LIN {X 0,Y 470.04,Z 195.084,A -85,B 0,C 180,E1 -7474.395,E2 -7474.395} C_VEL
LIN {X 0,Y 470.295,Z 182.109,A -85,B 0,C 180,E1 -7474.903,E2 -7474.903} C_VEL
LIN {X 0,Y 470.508,Z 169.126,A -85,B 0,C 180,E1 -7475.223,E2 -7475.223} C_VEL
LIN {X 0,Y 471.114,Z 78.667,A -85,B 0,C 180,E1 -7476.612,E2 -7476.612} C_VEL
LIN {X 0,Y 468.567,Z 65.779,A -85,B 0,C 180,E1 -7476.919,E2 -7476.919} C_VEL
LIN {X 0,Y 468.447,Z 59.054,A -85,B 0,C 180,E1 -7478.387,E2 -7478.387} C_VEL
LIN {X 0,Y 467.663,Z 54.233,A -85,B 0,C 180,E1 -7479.515,E2 -7479.515} C_VEL
LIN {X 0,Y 467.656,Z 54.231,A -85,B 0,C 180,E1 -7482.358,E2 -7482.358} C_VEL
LIN {X 0,Y 467.652,Z 54.229,A -85,B 0,C 180,E1 -7485.886,E2 -7485.886} C_VEL
LIN {X 0,Y 467.625,Z 54.231,A -85,B 0,C 180,E1 -7489.308,E2 -7489.308} C_VEL
LIN {X 0,Y 467.536,Z 54.247,A -85,B 0,C 180,E1 -7492.074,E2 -7492.074} C_VEL
LIN {X 0,Y 467.587,Z 54.237,A -85,B 0,C 180,E1 -7494.889,E2 -7494.889} C_VEL
LIN {X 0,Y 467.629,Z 54.234,A -85,B 0,C 180,E1 -7497.769,E2 -7497.769} C_VEL
LIN {X 0,Y 467.57,Z 54.238,A -85,B 0,C 180,E1 -7501.045,E2 -7501.045} C_VEL
LIN {X 0,Y 467.592,Z 54.238,A -85,B 0,C 180,E1 -7504.243,E2 -7504.243} C_VEL
LIN {X 0,Y 467.552,Z 54.242,A -85,B 0,C 180,E1 -7507.187,E2 -7507.187} C_VEL
LIN {X 0,Y 467.58,Z 54.238,A -85,B 0,C 180,E1 -7510.265,E2 -7510.265} C_VEL
LIN {X 0,Y 467.589,Z 54.236,A -85,B 0,C 180,E1 -7512.567,E2 -7512.567} C_VEL
LIN {X 0,Y 467.568,Z 54.241,A -85,B 0,C 180,E1 -7515.053,E2 -7515.053} C_VEL
LIN {X 0,Y 467.592,Z 54.243,A -85,B 0,C 180,E1 -7517.44,E2 -7517.44} C_VEL
LIN {X 0,Y 467.579,Z 54.24,A -85,B 0,C 180,E1 -7520.855,E2 -7520.855} C_VEL
LIN {X 0,Y 467.563,Z 54.239,A -85,B 0,C 180,E1 -7524.261,E2 -7524.261} C_VEL
LIN {X 0,Y 467.586,Z 54.24,A -85,B 0,C 180,E1 -7527.321,E2 -7527.321} C_VEL
LIN {X 0,Y 467.574,Z 54.242,A -85,B 0,C 180,E1 -7530.668,E2 -7530.668} C_VEL
LIN {X 0,Y 467.62,Z 54.235,A -85,B 0,C 180,E1 -7533.2,E2 -7533.2} C_VEL
LIN {X 0,Y 467.596,Z 54.24,A -85,B 0,C 180,E1 -7536.469,E2 -7536.469} C_VEL
LIN {X 0,Y 467.626,Z 54.231,A -85,B 0,C 180,E1 -7539.777,E2 -7539.777} C_VEL
LIN {X 0,Y 467.601,Z 54.242,A -85,B 0,C 180,E1 -7542.507,E2 -7542.507} C_VEL
LIN {X 0,Y 467.611,Z 54.233,A -85,B 0,C 180,E1 -7545.197,E2 -7545.197} C_VEL
LIN {X 0,Y 467.661,Z 54.229,A -85,B 0,C 180,E1 -7547.855,E2 -7547.855} C_VEL
LIN {X 0,Y 467.674,Z 54.225,A -85,B 0,C 180,E1 -7551.357,E2 -7551.357} C_VEL
LIN {X 0,Y 467.742,Z 54.223,A -85,B 0,C 180,E1 -7553.963,E2 -7553.963} C_VEL
LIN {X 0,Y 467.857,Z 54.204,A -85,B 0,C 180,E1 -7557.417,E2 -7557.417} C_VEL
LIN {X 0,Y 467.887,Z 54.205,A -85,B 0,C 180,E1 -7560,E2 -7560} C_VEL
LIN {X 0,Y 467.863,Z 54.202,A -85,B 0,C 180,E1 -7562.583,E2 -7562.583} C_VEL
LIN {X 0,Y 467.72,Z 54.222,A -85,B 0,C 180,E1 -7566.038,E2 -7566.038} C_VEL
LIN {X 0,Y 467.674,Z 54.225,A -85,B 0,C 180,E1 -7568.643,E2 -7568.643} C_VEL
LIN {X 0,Y 467.662,Z 54.227,A -85,B 0,C 180,E1 -7572.145,E2 -7572.145} C_VEL
LIN {X 0,Y 467.644,Z 54.232,A -85,B 0,C 180,E1 -7575.695,E2 -7575.695} C_VEL
LIN {X 0,Y 467.627,Z 54.237,A -85,B 0,C 180,E1 -7579.308,E2 -7579.308} C_VEL
LIN {X 0,Y 467.539,Z 54.242,A -85,B 0,C 180,E1 -7582.074,E2 -7582.074} C_VEL
LIN {X 0,Y 467.589,Z 54.243,A -85,B 0,C 180,E1 -7584.888,E2 -7584.888} C_VEL
LIN {X 0,Y 467.585,Z 54.236,A -85,B 0,C 180,E1 -7587.771,E2 -7587.771} C_VEL
LIN {X 0,Y 467.573,Z 54.242,A -85,B 0,C 180,E1 -7591.045,E2 -7591.045} C_VEL
LIN {X 0,Y 467.581,Z 54.24,A -85,B 0,C 180,E1 -7594.24,E2 -7594.24} C_VEL
LIN {X 0,Y 467.551,Z 54.241,A -85,B 0,C 180,E1 -7597.186,E2 -7597.186} C_VEL
LIN {X 0,Y 467.579,Z 54.243,A -85,B 0,C 180,E1 -7600.265,E2 -7600.265} C_VEL
LIN {X 0,Y 467.59,Z 54.24,A -85,B 0,C 180,E1 -7602.567,E2 -7602.567} C_VEL
LIN {X 0,Y 467.569,Z 54.238,A -85,B 0,C 180,E1 -7605.052,E2 -7605.052} C_VEL
LIN {X 0,Y 467.576,Z 54.239,A -85,B 0,C 180,E1 -7608.597,E2 -7608.597} C_VEL
LIN {X 0,Y 467.565,Z 54.247,A -85,B 0,C 180,E1 -7611.955,E2 -7611.955} C_VEL
LIN {X 0,Y 467.56,Z 54.24,A -85,B 0,C 180,E1 -7615.167,E2 -7615.167} C_VEL
LIN {X 0,Y 467.585,Z 54.238,A -85,B 0,C 180,E1 -7618.26,E2 -7618.26} C_VEL
LIN {X 0,Y 467.579,Z 54.243,A -85,B 0,C 180,E1 -7621.25,E2 -7621.25} C_VEL
LIN {X 0,Y 467.687,Z 54.395,A -85,B 0,C 180,E1 -7623.385,E2 -7623.385} C_VEL
LIN {X 0,Y 469.815,Z 65.941,A -85,B 0,C 180,E1 -7625.425,E2 -7625.425} C_VEL
LIN {X 0,Y 469.107,Z 85.156,A -85,B 0,C 180,E1 -7628.584,E2 -7628.584} C_VEL
LIN {X 0,Y 468.385,Z 105.335,A -85,B 0,C 180,E1 -7631.859,E2 -7631.859} C_VEL
LIN {X 0,Y 468.112,Z 112.972,A -85,B 0,C 180,E1 -7633.09,E2 -7633.09} C_VEL
LIN {X 0,Y 470.906,Z 134.248,A -85,B 0,C 180,E1 -7633.51,E2 -7633.51} C_VEL
LIN {X 0,Y 470.261,Z 221.943,A -85,B 0,C 180,E1 -7634.866,E2 -7634.866} C_VEL
LIN {X 0,Y 469.892,Z 235.212,A -85,B 0,C 180,E1 -7635.242,E2 -7635.242} C_VEL
LIN {X 0,Y 469.459,Z 247.401,A -85,B 0,C 180,E1 -7635.754,E2 -7635.754} C_VEL
LIN {X 0,Y 468.956,Z 259.7,A -85,B 0,C 180,E1 -7636.457,E2 -7636.457} C_VEL
LIN {X 0,Y 468.438,Z 270.965,A -85,B 0,C 180,E1 -7637.293,E2 -7637.293} C_VEL
LIN {X 0,Y 467.941,Z 281.832,A -85,B 0,C 180,E1 -7638.302,E2 -7638.302} C_VEL
LIN {X 0,Y 467.554,Z 291.258,A -85,B 0,C 180,E1 -7639.389,E2 -7639.389} C_VEL
LIN {X 0,Y 467.158,Z 300.369,A -85,B 0,C 180,E1 -7640.693,E2 -7640.693} C_VEL
LIN {X 0,Y 466.938,Z 307.713,A -85,B 0,C 180,E1 -7641.997,E2 -7641.997} C_VEL
LIN {X 0,Y 466.823,Z 312.679,A -85,B 0,C 180,E1 -7643.082,E2 -7643.082} C_VEL
LIN {X 0,Y 466.728,Z 317.498,A -85,B 0,C 180,E1 -7644.383,E2 -7644.383} C_VEL
LIN {X 0,Y 466.659,Z 321.185,A -85,B 0,C 180,E1 -7645.681,E2 -7645.681} C_VEL
LIN {X 0,Y 466.765,Z 323.097,A -85,B 0,C 180,E1 -7646.547,E2 -7646.547} C_VEL
LIN {X 0,Y 466.711,Z 324.536,A -85,B 0,C 180,E1 -7647.411,E2 -7647.411} C_VEL
LIN {X 0,Y 466.699,Z 325.556,A -85,B 0,C 180,E1 -7648.274,E2 -7648.274} C_VEL
LIN {X 0,Y 466.626,Z 326.42,A -85,B 0,C 180,E1 -7650,E2 -7650} C_VEL
LIN {X 0,Y 466.638,Z 326.234,A -85,B 0,C 180,E1 -7650.863,E2 -7650.863} C_VEL
LIN {X 0,Y 466.699,Z 325.64,A -85,B 0,C 180,E1 -7651.726,E2 -7651.726} C_VEL
LIN {X 0,Y 466.747,Z 323.273,A -85,B 0,C 180,E1 -7653.453,E2 -7653.453} C_VEL
LIN {X 0,Y 466.687,Z 320.35,A -85,B 0,C 180,E1 -7654.751,E2 -7654.751} C_VEL
LIN {X 0,Y 466.705,Z 316.398,A -85,B 0,C 180,E1 -7656.051,E2 -7656.051} C_VEL
LIN {X 0,Y 466.853,Z 311.32,A -85,B 0,C 180,E1 -7657.352,E2 -7657.352} C_VEL
LIN {X 0,Y 467.06,Z 304.951,A -85,B 0,C 180,E1 -7658.654,E2 -7658.654} C_VEL
LIN {X 0,Y 467.347,Z 296.995,A -85,B 0,C 180,E1 -7659.959,E2 -7659.959} C_VEL
LIN {X 0,Y 467.829,Z 288.916,A -85,B 0,C 180,E1 -7661.043,E2 -7661.043} C_VEL
LIN {X 0,Y 468.277,Z 279.075,A -85,B 0,C 180,E1 -7662.129,E2 -7662.129} C_VEL
LIN {X 0,Y 468.796,Z 268.113,A -85,B 0,C 180,E1 -7663.106,E2 -7663.106} C_VEL
LIN {X 0,Y 469.397,Z 255.626,A -85,B 0,C 180,E1 -7663.971,E2 -7663.971} C_VEL
LIN {X 0,Y 469.968,Z 243.381,A -85,B 0,C 180,E1 -7664.617,E2 -7664.617} C_VEL
LIN {X 0,Y 470.446,Z 230.499,A -85,B 0,C 180,E1 -7665.1,E2 -7665.1} C_VEL
LIN {X 0,Y 470.769,Z 216.847,A -85,B 0,C 180,E1 -7665.422,E2 -7665.422} C_VEL
LIN {X 0,Y 471.263,Z 132.801,A -85,B 0,C 180,E1 -7666.727,E2 -7666.727} C_VEL
LIN {X 0,Y 468.293,Z 112.618,A -85,B 0,C 180,E1 -7667.179,E2 -7667.179} C_VEL
LIN {X 0,Y 469.033,Z 94.5,A -85,B 0,C 180,E1 -7670.159,E2 -7670.159} C_VEL
LIN {X 0,Y 469.874,Z 75.402,A -85,B 0,C 180,E1 -7673.351,E2 -7673.351} C_VEL
LIN {X 0,Y 470.248,Z 67.22,A -85,B 0,C 180,E1 -7674.738,E2 -7674.738} C_VEL
LIN {X 0,Y 468.091,Z 56.28,A -85,B 0,C 180,E1 -7676.771,E2 -7676.771} C_VEL
LIN {X 0,Y 467.673,Z 54.232,A -85,B 0,C 180,E1 -7677.19,E2 -7677.19} C_VEL
LIN {X 0,Y 467.572,Z 54.239,A -85,B 0,C 180,E1 -7680.734,E2 -7680.734} C_VEL
LIN {X 0,Y 467.572,Z 54.244,A -85,B 0,C 180,E1 -7683.79,E2 -7683.79} C_VEL
LIN {X 0,Y 467.532,Z 54.244,A -85,B 0,C 180,E1 -7686.962,E2 -7686.962} C_VEL
LIN {X 0,Y 467.585,Z 54.237,A -85,B 0,C 180,E1 -7689.955,E2 -7689.955} C_VEL
LIN {X 0,Y 467.589,Z 54.235,A -85,B 0,C 180,E1 -7692.567,E2 -7692.567} C_VEL
LIN {X 0,Y 467.569,Z 54.237,A -85,B 0,C 180,E1 -7695.053,E2 -7695.053} C_VEL
LIN {X 0,Y 467.592,Z 54.238,A -85,B 0,C 180,E1 -7697.44,E2 -7697.44} C_VEL
LIN {X 0,Y 467.563,Z 54.237,A -85,B 0,C 180,E1 -7700.853,E2 -7700.853} C_VEL
LIN {X 0,Y 467.562,Z 54.238,A -85,B 0,C 180,E1 -7704.261,E2 -7704.261} C_VEL
LIN {X 0,Y 467.583,Z 54.243,A -85,B 0,C 180,E1 -7707.321,E2 -7707.321} C_VEL
LIN {X 0,Y 467.574,Z 54.239,A -85,B 0,C 180,E1 -7710.667,E2 -7710.667} C_VEL
LIN {X 0,Y 467.619,Z 54.234,A -85,B 0,C 180,E1 -7713.2,E2 -7713.2} C_VEL
LIN {X 0,Y 467.596,Z 54.239,A -85,B 0,C 180,E1 -7716.468,E2 -7716.468} C_VEL
LIN {X 0,Y 467.626,Z 54.231,A -85,B 0,C 180,E1 -7719.777,E2 -7719.777} C_VEL
LIN {X 0,Y 467.61,Z 54.236,A -85,B 0,C 180,E1 -7722.507,E2 -7722.507} C_VEL
LIN {X 0,Y 467.611,Z 54.234,A -85,B 0,C 180,E1 -7725.196,E2 -7725.196} C_VEL
LIN {X 0,Y 467.661,Z 54.226,A -85,B 0,C 180,E1 -7727.855,E2 -7727.855} C_VEL
LIN {X 0,Y 467.685,Z 54.225,A -85,B 0,C 180,E1 -7731.357,E2 -7731.357} C_VEL
LIN {X 0,Y 467.742,Z 54.218,A -85,B 0,C 180,E1 -7733.962,E2 -7733.962} C_VEL
LIN {X 0,Y 467.856,Z 54.204,A -85,B 0,C 180,E1 -7737.417,E2 -7737.417} C_VEL
LIN {X 0,Y 467.886,Z 54.205,A -85,B 0,C 180,E1 -7740,E2 -7740} C_VEL
LIN {X 0,Y 467.862,Z 54.2,A -85,B 0,C 180,E1 -7742.583,E2 -7742.583} C_VEL
LIN {X 0,Y 467.73,Z 54.221,A -85,B 0,C 180,E1 -7746.037,E2 -7746.037} C_VEL
LIN {X 0,Y 467.673,Z 54.222,A -85,B 0,C 180,E1 -7748.643,E2 -7748.643} C_VEL
LIN {X 0,Y 467.66,Z 54.227,A -85,B 0,C 180,E1 -7752.145,E2 -7752.145} C_VEL
LIN {X 0,Y 467.643,Z 54.232,A -85,B 0,C 180,E1 -7755.695,E2 -7755.695} C_VEL
LIN {X 0,Y 467.625,Z 54.236,A -85,B 0,C 180,E1 -7759.308,E2 -7759.308} C_VEL
LIN {X 0,Y 467.538,Z 54.242,A -85,B 0,C 180,E1 -7762.074,E2 -7762.074} C_VEL
LIN {X 0,Y 467.595,Z 54.243,A -85,B 0,C 180,E1 -7764.888,E2 -7764.888} C_VEL
LIN {X 0,Y 467.583,Z 54.236,A -85,B 0,C 180,E1 -7767.771,E2 -7767.771} C_VEL
LIN {X 0,Y 467.571,Z 54.24,A -85,B 0,C 180,E1 -7771.045,E2 -7771.045} C_VEL
LIN {X 0,Y 467.579,Z 54.241,A -85,B 0,C 180,E1 -7774.24,E2 -7774.24} C_VEL
LIN {X 0,Y 467.545,Z 54.241,A -85,B 0,C 180,E1 -7777.185,E2 -7777.185} C_VEL
LIN {X 0,Y 467.571,Z 54.237,A -85,B 0,C 180,E1 -7780.265,E2 -7780.265} C_VEL
LIN {X 0,Y 467.55,Z 54.247,A -85,B 0,C 180,E1 -7783.745,E2 -7783.745} C_VEL
LIN {X 0,Y 467.549,Z 54.247,A -85,B 0,C 180,E1 -7786.255,E2 -7786.255} C_VEL
LIN {X 0,Y 467.576,Z 54.24,A -85,B 0,C 180,E1 -7788.724,E2 -7788.724} C_VEL
LIN {X 0,Y 467.562,Z 54.246,A -85,B 0,C 180,E1 -7791.955,E2 -7791.955} C_VEL
LIN {X 0,Y 467.558,Z 54.246,A -85,B 0,C 180,E1 -7795.167,E2 -7795.167} C_VEL
LIN {X 0,Y 467.583,Z 54.245,A -85,B 0,C 180,E1 -7798.26,E2 -7798.26} C_VEL
LIN {X 0,Y 467.654,Z 54.399,A -85,B 0,C 180,E1 -7800.207,E2 -7800.207} C_VEL
LIN {X 0,Y 468.798,Z 61.23,A -85,B 0,C 180,E1 -7801.811,E2 -7801.811} C_VEL
LIN {X 0,Y 468.782,Z 66.257,A -85,B 0,C 180,E1 -7802.91,E2 -7802.91} C_VEL
LIN {X 0,Y 471.756,Z 79.365,A -85,B 0,C 180,E1 -7803.245,E2 -7803.245} C_VEL
LIN {X 0,Y 471.132,Z 151.793,A -85,B 0,C 180,E1 -7804.364,E2 -7804.364} C_VEL
LIN {X 0,Y 470.45,Z 157.646,A -85,B 0,C 180,E1 -7804.426,E2 -7804.426} C_VEL
LIN {X 0,Y 464.651,Z 176.593,A -85,B 0,C 180,E1 -7804.553,E2 -7804.553} C_VEL
LIN {X 0,Y 464.096,Z 180.421,A -85,B 0,C 180,E1 -7804.641,E2 -7804.641} C_VEL
LIN {X 0,Y 464.057,Z 182.332,A -85,B 0,C 180,E1 -7804.7,E2 -7804.7} C_VEL
LIN {X 0,Y 463.797,Z 194.305,A -85,B 0,C 180,E1 -7805.165,E2 -7805.165} C_VEL
LIN {X 0,Y 463.318,Z 206.546,A -85,B 0,C 180,E1 -7805.823,E2 -7805.823} C_VEL
LIN {X 0,Y 462.778,Z 217.982,A -85,B 0,C 180,E1 -7806.625,E2 -7806.625} C_VEL
LIN {X 0,Y 462.245,Z 228.376,A -85,B 0,C 180,E1 -7807.542,E2 -7807.542} C_VEL
LIN {X 0,Y 461.773,Z 237.821,A -85,B 0,C 180,E1 -7808.576,E2 -7808.576} C_VEL
LIN {X 0,Y 461.235,Z 246.36,A -85,B 0,C 180,E1 -7809.717,E2 -7809.717} C_VEL
LIN {X 0,Y 460.738,Z 254.387,A -85,B 0,C 180,E1 -7811.038,E2 -7811.038} C_VEL
LIN {X 0,Y 460.447,Z 260.231,A -85,B 0,C 180,E1 -7812.226,E2 -7812.226} C_VEL
LIN {X 0,Y 460.138,Z 265.635,A -85,B 0,C 180,E1 -7813.587,E2 -7813.587} C_VEL
LIN {X 0,Y 459.936,Z 269.802,A -85,B 0,C 180,E1 -7814.944,E2 -7814.944} C_VEL
LIN {X 0,Y 459.797,Z 271.963,A -85,B 0,C 180,E1 -7815.844,E2 -7815.844} C_VEL
LIN {X 0,Y 459.717,Z 273.644,A -85,B 0,C 180,E1 -7816.743,E2 -7816.743} C_VEL
LIN {X 0,Y 459.659,Z 275.394,A -85,B 0,C 180,E1 -7818.107,E2 -7818.107} C_VEL
LIN {X 0,Y 459.611,Z 276.18,A -85,B 0,C 180,E1 -7819.427,E2 -7819.427} C_VEL
LIN {X 0,Y 459.606,Z 275.831,A -85,B 0,C 180,E1 -7821.204,E2 -7821.204} C_VEL
LIN {X 0,Y 459.657,Z 275.064,A -85,B 0,C 180,E1 -7822.091,E2 -7822.091} C_VEL
LIN {X 0,Y 459.784,Z 272.99,A -85,B 0,C 180,E1 -7823.491,E2 -7823.491} C_VEL
LIN {X 0,Y 459.811,Z 270.242,A -85,B 0,C 180,E1 -7824.738,E2 -7824.738} C_VEL
LIN {X 0,Y 460.024,Z 266.325,A -85,B 0,C 180,E1 -7826.058,E2 -7826.058} C_VEL
LIN {X 0,Y 460.127,Z 261.308,A -85,B 0,C 180,E1 -7827.374,E2 -7827.374} C_VEL
LIN {X 0,Y 460.461,Z 254.977,A -85,B 0,C 180,E1 -7828.688,E2 -7828.688} C_VEL
LIN {X 0,Y 460.855,Z 247.091,A -85,B 0,C 180,E1 -7830,E2 -7830} C_VEL
LIN {X 0,Y 461.294,Z 237.315,A -85,B 0,C 180,E1 -7831.31,E2 -7831.31} C_VEL
LIN {X 0,Y 461.816,Z 228.201,A -85,B 0,C 180,E1 -7832.29,E2 -7832.29} C_VEL
LIN {X 0,Y 462.324,Z 218.3,A -85,B 0,C 180,E1 -7833.159,E2 -7833.159} C_VEL
LIN {X 0,Y 462.804,Z 207.555,A -85,B 0,C 180,E1 -7833.918,E2 -7833.918} C_VEL
LIN {X 0,Y 463.122,Z 195.771,A -85,B 0,C 180,E1 -7834.57,E2 -7834.57} C_VEL
LIN {X 0,Y 463.393,Z 182.979,A -85,B 0,C 180,E1 -7835.085,E2 -7835.085} C_VEL
LIN {X 0,Y 463.614,Z 170.316,A -85,B 0,C 180,E1 -7835.409,E2 -7835.409} C_VEL
LIN {X 0,Y 464.301,Z 79.935,A -85,B 0,C 180,E1 -7836.819,E2 -7836.819} C_VEL
LIN {X 0,Y 461.608,Z 66.201,A -85,B 0,C 180,E1 -7837.133,E2 -7837.133} C_VEL
LIN {X 0,Y 461.454,Z 60.029,A -85,B 0,C 180,E1 -7838.496,E2 -7838.496} C_VEL
LIN {X 0,Y 460.612,Z 55.112,A -85,B 0,C 180,E1 -7839.662,E2 -7839.662} C_VEL
LIN {X 0,Y 460.615,Z 55.11,A -85,B 0,C 180,E1 -7842.445,E2 -7842.445} C_VEL
LIN {X 0,Y 460.602,Z 55.108,A -85,B 0,C 180,E1 -7845.998,E2 -7845.998} C_VEL
LIN {X 0,Y 460.573,Z 55.112,A -85,B 0,C 180,E1 -7848.902,E2 -7848.902} C_VEL
LIN {X 0,Y 460.518,Z 55.117,A -85,B 0,C 180,E1 -7851.486,E2 -7851.486} C_VEL
LIN {X 0,Y 460.533,Z 55.121,A -85,B 0,C 180,E1 -7854.333,E2 -7854.333} C_VEL
LIN {X 0,Y 460.591,Z 55.111,A -85,B 0,C 180,E1 -7857.748,E2 -7857.748} C_VEL
LIN {X 0,Y 460.523,Z 55.117,A -85,B 0,C 180,E1 -7861.283,E2 -7861.283} C_VEL
LIN {X 0,Y 460.536,Z 55.115,A -85,B 0,C 180,E1 -7864.506,E2 -7864.506} C_VEL
LIN {X 0,Y 460.53,Z 55.121,A -85,B 0,C 180,E1 -7867.621,E2 -7867.621} C_VEL
LIN {X 0,Y 460.544,Z 55.114,A -85,B 0,C 180,E1 -7870.27,E2 -7870.27} C_VEL
LIN {X 0,Y 460.501,Z 55.124,A -85,B 0,C 180,E1 -7873.376,E2 -7873.376} C_VEL
LIN {X 0,Y 460.501,Z 55.119,A -85,B 0,C 180,E1 -7876.625,E2 -7876.625} C_VEL
LIN {X 0,Y 460.542,Z 55.116,A -85,B 0,C 180,E1 -7879.731,E2 -7879.731} C_VEL
LIN {X 0,Y 460.503,Z 55.119,A -85,B 0,C 180,E1 -7882.524,E2 -7882.524} C_VEL
LIN {X 0,Y 460.55,Z 55.114,A -85,B 0,C 180,E1 -7885.624,E2 -7885.624} C_VEL
LIN {X 0,Y 460.541,Z 55.119,A -85,B 0,C 180,E1 -7888.745,E2 -7888.745} C_VEL
LIN {X 0,Y 460.585,Z 55.109,A -85,B 0,C 180,E1 -7892.254,E2 -7892.254} C_VEL
LIN {X 0,Y 460.562,Z 55.118,A -85,B 0,C 180,E1 -7894.706,E2 -7894.706} C_VEL
LIN {X 0,Y 460.515,Z 55.117,A -85,B 0,C 180,E1 -7897.572,E2 -7897.572} C_VEL
LIN {X 0,Y 460.572,Z 55.115,A -85,B 0,C 180,E1 -7900.385,E2 -7900.385} C_VEL
LIN {X 0,Y 460.609,Z 55.109,A -85,B 0,C 180,E1 -7904.059,E2 -7904.059} C_VEL
LIN {X 0,Y 460.614,Z 55.106,A -85,B 0,C 180,E1 -7907.666,E2 -7907.666} C_VEL
LIN {X 0,Y 460.624,Z 55.103,A -85,B 0,C 180,E1 -7911.224,E2 -7911.224} C_VEL
LIN {X 0,Y 460.707,Z 55.098,A -85,B 0,C 180,E1 -7913.87,E2 -7913.87} C_VEL
LIN {X 0,Y 460.797,Z 55.083,A -85,B 0,C 180,E1 -7917.378,E2 -7917.378} C_VEL
LIN {X 0,Y 460.858,Z 55.08,A -85,B 0,C 180,E1 -7920,E2 -7920} C_VEL
LIN {X 0,Y 460.804,Z 55.081,A -85,B 0,C 180,E1 -7922.623,E2 -7922.623} C_VEL
LIN {X 0,Y 460.685,Z 55.098,A -85,B 0,C 180,E1 -7926.13,E2 -7926.13} C_VEL
LIN {X 0,Y 460.624,Z 55.104,A -85,B 0,C 180,E1 -7928.776,E2 -7928.776} C_VEL
LIN {X 0,Y 460.619,Z 55.104,A -85,B 0,C 180,E1 -7932.445,E2 -7932.445} C_VEL
LIN {X 0,Y 460.606,Z 55.106,A -85,B 0,C 180,E1 -7935.997,E2 -7935.997} C_VEL
LIN {X 0,Y 460.573,Z 55.112,A -85,B 0,C 180,E1 -7939.615,E2 -7939.615} C_VEL
LIN {X 0,Y 460.515,Z 55.118,A -85,B 0,C 180,E1 -7942.429,E2 -7942.429} C_VEL
LIN {X 0,Y 460.553,Z 55.112,A -85,B 0,C 180,E1 -7945.797,E2 -7945.797} C_VEL
LIN {X 0,Y 460.532,Z 55.116,A -85,B 0,C 180,E1 -7948.235,E2 -7948.235} C_VEL
LIN {X 0,Y 460.525,Z 55.117,A -85,B 0,C 180,E1 -7951.283,E2 -7951.283} C_VEL
LIN {X 0,Y 460.527,Z 55.122,A -85,B 0,C 180,E1 -7954.504,E2 -7954.504} C_VEL
LIN {X 0,Y 460.505,Z 55.118,A -85,B 0,C 180,E1 -7957.623,E2 -7957.623} C_VEL
LIN {X 0,Y 460.543,Z 55.12,A -85,B 0,C 180,E1 -7960.269,E2 -7960.269} C_VEL
LIN {X 0,Y 460.5,Z 55.119,A -85,B 0,C 180,E1 -7963.376,E2 -7963.376} C_VEL
LIN {X 0,Y 460.512,Z 55.12,A -85,B 0,C 180,E1 -7966.625,E2 -7966.625} C_VEL
LIN {X 0,Y 460.538,Z 55.118,A -85,B 0,C 180,E1 -7969.732,E2 -7969.732} C_VEL
LIN {X 0,Y 460.5,Z 55.12,A -85,B 0,C 180,E1 -7972.524,E2 -7972.524} C_VEL
LIN {X 0,Y 460.54,Z 55.119,A -85,B 0,C 180,E1 -7975.623,E2 -7975.623} C_VEL
LIN {X 0,Y 460.541,Z 55.114,A -85,B 0,C 180,E1 -7978.744,E2 -7978.744} C_VEL
LIN {X 0,Y 460.585,Z 55.113,A -85,B 0,C 180,E1 -7982.254,E2 -7982.254} C_VEL
LIN {X 0,Y 460.657,Z 55.196,A -85,B 0,C 180,E1 -7983.191,E2 -7983.191} C_VEL
LIN {X 0,Y 462.874,Z 67.26,A -85,B 0,C 180,E1 -7985.356,E2 -7985.356} C_VEL
LIN {X 0,Y 462.084,Z 86.657,A -85,B 0,C 180,E1 -7988.591,E2 -7988.591} C_VEL
LIN {X 0,Y 461.359,Z 106.149,A -85,B 0,C 180,E1 -7991.803,E2 -7991.803} C_VEL
LIN {X 0,Y 461.112,Z 112.556,A -85,B 0,C 180,E1 -7992.852,E2 -7992.852} C_VEL
LIN {X 0,Y 464.049,Z 134.854,A -85,B 0,C 180,E1 -7993.304,E2 -7993.304} C_VEL
LIN {X 0,Y 463.377,Z 221.566,A -85,B 0,C 180,E1 -7994.664,E2 -7994.664} C_VEL
LIN {X 0,Y 462.968,Z 234.835,A -85,B 0,C 180,E1 -7995.045,E2 -7995.045} C_VEL
LIN {X 0,Y 462.499,Z 247.596,A -85,B 0,C 180,E1 -7995.592,E2 -7995.592} C_VEL
LIN {X 0,Y 462.024,Z 258.932,A -85,B 0,C 180,E1 -7996.25,E2 -7996.25} C_VEL
LIN {X 0,Y 461.492,Z 269.96,A -85,B 0,C 180,E1 -7997.072,E2 -7997.072} C_VEL
LIN {X 0,Y 460.934,Z 281.194,A -85,B 0,C 180,E1 -7998.121,E2 -7998.121} C_VEL
LIN {X 0,Y 460.547,Z 290.685,A -85,B 0,C 180,E1 -7999.226,E2 -7999.226} C_VEL
LIN {X 0,Y 460.118,Z 299.831,A -85,B 0,C 180,E1 -8000.549,E2 -8000.549} C_VEL
LIN {X 0,Y 459.884,Z 307.206,A -85,B 0,C 180,E1 -8001.873,E2 -8001.873} C_VEL
LIN {X 0,Y 459.734,Z 312.195,A -85,B 0,C 180,E1 -8002.975,E2 -8002.975} C_VEL
LIN {X 0,Y 459.622,Z 317.037,A -85,B 0,C 180,E1 -8004.296,E2 -8004.296} C_VEL
LIN {X 0,Y 459.574,Z 320.745,A -85,B 0,C 180,E1 -8005.615,E2 -8005.615} C_VEL
LIN {X 0,Y 459.673,Z 322.666,A -85,B 0,C 180,E1 -8006.494,E2 -8006.494} C_VEL
LIN {X 0,Y 459.632,Z 324.124,A -85,B 0,C 180,E1 -8007.371,E2 -8007.371} C_VEL
LIN {X 0,Y 459.635,Z 325.153,A -85,B 0,C 180,E1 -8008.247,E2 -8008.247} C_VEL
LIN {X 0,Y 459.556,Z 326.033,A -85,B 0,C 180,E1 -8010,E2 -8010} C_VEL
LIN {X 0,Y 459.57,Z 325.862,A -85,B 0,C 180,E1 -8010.876,E2 -8010.876} C_VEL
LIN {X 0,Y 459.606,Z 325.275,A -85,B 0,C 180,E1 -8011.752,E2 -8011.752} C_VEL
LIN {X 0,Y 459.631,Z 324.298,A -85,B 0,C 180,E1 -8012.629,E2 -8012.629} C_VEL
LIN {X 0,Y 459.641,Z 322.923,A -85,B 0,C 180,E1 -8013.506,E2 -8013.506} C_VEL
LIN {X 0,Y 459.613,Z 320.02,A -85,B 0,C 180,E1 -8014.824,E2 -8014.824} C_VEL
LIN {X 0,Y 459.635,Z 315.42,A -85,B 0,C 180,E1 -8016.342,E2 -8016.342} C_VEL
LIN {X 0,Y 459.862,Z 309.054,A -85,B 0,C 180,E1 -8017.906,E2 -8017.906} C_VEL
LIN {X 0,Y 460.081,Z 302.225,A -85,B 0,C 180,E1 -8019.23,E2 -8019.23} C_VEL
LIN {X 0,Y 460.47,Z 293.763,A -85,B 0,C 180,E1 -8020.553,E2 -8020.553} C_VEL
LIN {X 0,Y 460.991,Z 285.07,A -85,B 0,C 180,E1 -8021.654,E2 -8021.654} C_VEL
LIN {X 0,Y 461.533,Z 274.017,A -85,B 0,C 180,E1 -8022.791,E2 -8022.791} C_VEL
LIN {X 0,Y 462.12,Z 263.799,A -85,B 0,C 180,E1 -8023.635,E2 -8023.635} C_VEL
LIN {X 0,Y 462.745,Z 252.029,A -85,B 0,C 180,E1 -8024.401,E2 -8024.401} C_VEL
LIN {X 0,Y 463.296,Z 239.822,A -85,B 0,C 180,E1 -8025.001,E2 -8025.001} C_VEL
LIN {X 0,Y 463.755,Z 227.405,A -85,B 0,C 180,E1 -8025.435,E2 -8025.435} C_VEL
LIN {X 0,Y 463.99,Z 214.988,A -85,B 0,C 180,E1 -8025.709,E2 -8025.709} C_VEL
LIN {X 0,Y 464.578,Z 133.953,A -85,B 0,C 180,E1 -8026.981,E2 -8026.981} C_VEL
LIN {X 0,Y 461.333,Z 112.253,A -85,B 0,C 180,E1 -8027.473,E2 -8027.473} C_VEL
LIN {X 0,Y 462.067,Z 95.691,A -85,B 0,C 180,E1 -8030.245,E2 -8030.245} C_VEL
LIN {X 0,Y 462.827,Z 79.337,A -85,B 0,C 180,E1 -8033.018,E2 -8033.018} C_VEL
LIN {X 0,Y 463.369,Z 69.35,A -85,B 0,C 180,E1 -8034.732,E2 -8034.732} C_VEL
LIN {X 0,Y 461.754,Z 60.249,A -85,B 0,C 180,E1 -8036.436,E2 -8036.436} C_VEL
LIN {X 0,Y 460.619,Z 55.111,A -85,B 0,C 180,E1 -8037.448,E2 -8037.448} C_VEL
LIN {X 0,Y 460.513,Z 55.122,A -85,B 0,C 180,E1 -8040.24,E2 -8040.24} C_VEL
LIN {X 0,Y 460.522,Z 55.119,A -85,B 0,C 180,E1 -8043.326,E2 -8043.326} C_VEL
LIN {X 0,Y 460.479,Z 55.125,A -85,B 0,C 180,E1 -8046.529,E2 -8046.529} C_VEL
LIN {X 0,Y 460.535,Z 55.114,A -85,B 0,C 180,E1 -8049.862,E2 -8049.862} C_VEL
LIN {X 0,Y 460.515,Z 55.116,A -85,B 0,C 180,E1 -8052.9,E2 -8052.9} C_VEL
LIN {X 0,Y 460.512,Z 55.121,A -85,B 0,C 180,E1 -8055.831,E2 -8055.831} C_VEL
LIN {X 0,Y 460.534,Z 55.115,A -85,B 0,C 180,E1 -8058.989,E2 -8058.989} C_VEL
LIN {X 0,Y 460.522,Z 55.119,A -85,B 0,C 180,E1 -8061.266,E2 -8061.266} C_VEL
LIN {X 0,Y 460.512,Z 55.117,A -85,B 0,C 180,E1 -8064.554,E2 -8064.554} C_VEL
LIN {X 0,Y 460.533,Z 55.117,A -85,B 0,C 180,E1 -8067.716,E2 -8067.716} C_VEL
LIN {X 0,Y 460.544,Z 55.115,A -85,B 0,C 180,E1 -8070.769,E2 -8070.769} C_VEL
LIN {X 0,Y 460.563,Z 55.109,A -85,B 0,C 180,E1 -8073.735,E2 -8073.735} C_VEL
LIN {X 0,Y 460.549,Z 55.119,A -85,B 0,C 180,E1 -8076.624,E2 -8076.624} C_VEL
LIN {X 0,Y 460.555,Z 55.112,A -85,B 0,C 180,E1 -8079.453,E2 -8079.453} C_VEL
LIN {X 0,Y 460.562,Z 55.115,A -85,B 0,C 180,E1 -8082.23,E2 -8082.23} C_VEL
LIN {X 0,Y 460.57,Z 55.113,A -85,B 0,C 180,E1 -8084.965,E2 -8084.965} C_VEL
LIN {X 0,Y 460.615,Z 55.108,A -85,B 0,C 180,E1 -8088.559,E2 -8088.559} C_VEL
LIN {X 0,Y 460.7,Z 55.097,A -85,B 0,C 180,E1 -8092.108,E2 -8092.108} C_VEL
LIN {X 0,Y 460.699,Z 55.095,A -85,B 0,C 180,E1 -8094.748,E2 -8094.748} C_VEL
LIN {X 0,Y 460.797,Z 55.083,A -85,B 0,C 180,E1 -8097.377,E2 -8097.377} C_VEL
LIN {X 0,Y 460.857,Z 55.081,A -85,B 0,C 180,E1 -8100,E2 -8100} C_VEL
LIN {X 0,Y 460.802,Z 55.079,A -85,B 0,C 180,E1 -8102.622,E2 -8102.622} C_VEL
LIN {X 0,Y 460.696,Z 55.097,A -85,B 0,C 180,E1 -8106.13,E2 -8106.13} C_VEL
LIN {X 0,Y 460.623,Z 55.101,A -85,B 0,C 180,E1 -8108.776,E2 -8108.776} C_VEL
LIN {X 0,Y 460.617,Z 55.105,A -85,B 0,C 180,E1 -8112.445,E2 -8112.445} C_VEL
LIN {X 0,Y 460.604,Z 55.107,A -85,B 0,C 180,E1 -8115.997,E2 -8115.997} C_VEL
LIN {X 0,Y 460.571,Z 55.111,A -85,B 0,C 180,E1 -8119.615,E2 -8119.615} C_VEL
LIN {X 0,Y 460.514,Z 55.119,A -85,B 0,C 180,E1 -8122.428,E2 -8122.428} C_VEL
LIN {X 0,Y 460.552,Z 55.113,A -85,B 0,C 180,E1 -8125.797,E2 -8125.797} C_VEL
LIN {X 0,Y 460.53,Z 55.117,A -85,B 0,C 180,E1 -8128.234,E2 -8128.234} C_VEL
LIN {X 0,Y 460.523,Z 55.117,A -85,B 0,C 180,E1 -8131.283,E2 -8131.283} C_VEL
LIN {X 0,Y 460.524,Z 55.121,A -85,B 0,C 180,E1 -8134.503,E2 -8134.503} C_VEL
LIN {X 0,Y 460.5,Z 55.12,A -85,B 0,C 180,E1 -8137.623,E2 -8137.623} C_VEL
LIN {X 0,Y 460.528,Z 55.11,A -85,B 0,C 180,E1 -8141.012,E2 -8141.012} C_VEL
LIN {X 0,Y 460.514,Z 55.121,A -85,B 0,C 180,E1 -8144.589,E2 -8144.589} C_VEL
LIN {X 0,Y 460.505,Z 55.125,A -85,B 0,C 180,E1 -8147.816,E2 -8147.816} C_VEL
LIN {X 0,Y 460.519,Z 55.122,A -85,B 0,C 180,E1 -8150.136,E2 -8150.136} C_VEL
LIN {X 0,Y 460.473,Z 55.13,A -85,B 0,C 180,E1 -8153.47,E2 -8153.47} C_VEL
LIN {X 0,Y 460.521,Z 55.123,A -85,B 0,C 180,E1 -8156.674,E2 -8156.674} C_VEL
LIN {X 0,Y 460.591,Z 55.305,A -85,B 0,C 180,E1 -8159.983,E2 -8159.983} C_VEL
LIN {X 0,Y 461.913,Z 63.182,A -85,B 0,C 180,E1 -8161.857,E2 -8161.857} C_VEL
LIN {X 0,Y 461.881,Z 66.521,A -85,B 0,C 180,E1 -8162.606,E2 -8162.606} C_VEL
LIN {X 0,Y 465.099,Z 80.549,A -85,B 0,C 180,E1 -8162.979,E2 -8162.979} C_VEL
LIN {X 0,Y 464.19,Z 172.656,A -85,B 0,C 180,E1 -8164.437,E2 -8164.437} C_VEL
LIN {X 0,Y 464.057,Z 182.332,A -85,B 0,C 180,E1 -8164.7,E2 -8164.7} C_VEL
LIN {X 0,Y 463.383,Z 188.041,A -85,B 0,C 180,E1 -8164.872,E2 -8164.872} C_VEL
LIN {X 0,Y 460.395,Z 197.222,A -85,B 0,C 180,E1 -8165.158,E2 -8165.158} C_VEL
LIN {X 0,Y 457.24,Z 206.104,A -85,B 0,C 180,E1 -8165.542,E2 -8165.542} C_VEL
LIN {X 0,Y 456.311,Z 211.34,A -85,B 0,C 180,E1 -8165.863,E2 -8165.863} C_VEL
LIN {X 0,Y 455.712,Z 222.361,A -85,B 0,C 180,E1 -8166.722,E2 -8166.722} C_VEL
LIN {X 0,Y 455.12,Z 233.364,A -85,B 0,C 180,E1 -8167.802,E2 -8167.802} C_VEL
LIN {X 0,Y 454.571,Z 242.586,A -85,B 0,C 180,E1 -8168.933,E2 -8168.933} C_VEL
LIN {X 0,Y 453.992,Z 251.719,A -85,B 0,C 180,E1 -8170.322,E2 -8170.322} C_VEL
LIN {X 0,Y 453.531,Z 259.009,A -85,B 0,C 180,E1 -8171.712,E2 -8171.712} C_VEL
LIN {X 0,Y 453.233,Z 263.882,A -85,B 0,C 180,E1 -8172.865,E2 -8172.865} C_VEL
LIN {X 0,Y 452.994,Z 268.211,A -85,B 0,C 180,E1 -8174.134,E2 -8174.134} C_VEL
LIN {X 0,Y 452.758,Z 272.079,A -85,B 0,C 180,E1 -8175.619,E2 -8175.619} C_VEL
LIN {X 0,Y 452.666,Z 273.822,A -85,B 0,C 180,E1 -8176.533,E2 -8176.533} C_VEL
LIN {X 0,Y 452.573,Z 275.781,A -85,B 0,C 180,E1 -8178.049,E2 -8178.049} C_VEL
LIN {X 0,Y 452.552,Z 276.542,A -85,B 0,C 180,E1 -8179.26,E2 -8179.26} C_VEL
LIN {X 0,Y 452.508,Z 276.286,A -85,B 0,C 180,E1 -8181.065,E2 -8181.065} C_VEL
LIN {X 0,Y 452.554,Z 275.577,A -85,B 0,C 180,E1 -8181.966,E2 -8181.966} C_VEL
LIN {X 0,Y 452.696,Z 273.392,A -85,B 0,C 180,E1 -8183.507,E2 -8183.507} C_VEL
LIN {X 0,Y 452.752,Z 269.774,A -85,B 0,C 180,E1 -8185.102,E2 -8185.102} C_VEL
LIN {X 0,Y 452.999,Z 265.598,A -85,B 0,C 180,E1 -8186.442,E2 -8186.442} C_VEL
LIN {X 0,Y 453.185,Z 259.281,A -85,B 0,C 180,E1 -8188,E2 -8188} C_VEL
LIN {X 0,Y 453.614,Z 252.377,A -85,B 0,C 180,E1 -8189.334,E2 -8189.334} C_VEL
LIN {X 0,Y 454.002,Z 243.76,A -85,B 0,C 180,E1 -8190.665,E2 -8190.665} C_VEL
LIN {X 0,Y 454.448,Z 234.945,A -85,B 0,C 180,E1 -8191.773,E2 -8191.773} C_VEL
LIN {X 0,Y 454.978,Z 225.255,A -85,B 0,C 180,E1 -8192.767,E2 -8192.767} C_VEL
LIN {X 0,Y 455.54,Z 214.598,A -85,B 0,C 180,E1 -8193.649,E2 -8193.649} C_VEL
LIN {X 0,Y 455.996,Z 202.692,A -85,B 0,C 180,E1 -8194.42,E2 -8194.42} C_VEL
LIN {X 0,Y 456.358,Z 190.303,A -85,B 0,C 180,E1 -8195.025,E2 -8195.025} C_VEL
LIN {X 0,Y 456.614,Z 177.301,A -85,B 0,C 180,E1 -8195.465,E2 -8195.465} C_VEL
LIN {X 0,Y 456.805,Z 161.64,A -85,B 0,C 180,E1 -8195.767,E2 -8195.767} C_VEL
LIN {X 0,Y 457.353,Z 80.446,A -85,B 0,C 180,E1 -8197.046,E2 -8197.046} C_VEL
LIN {X 0,Y 454.655,Z 66.487,A -85,B 0,C 180,E1 -8197.383,E2 -8197.383} C_VEL
LIN {X 0,Y 454.51,Z 61.595,A -85,B 0,C 180,E1 -8198.474,E2 -8198.474} C_VEL
LIN {X 0,Y 453.573,Z 55.988,A -85,B 0,C 180,E1 -8199.814,E2 -8199.814} C_VEL
LIN {X 0,Y 453.565,Z 55.989,A -85,B 0,C 180,E1 -8202.529,E2 -8202.529} C_VEL
LIN {X 0,Y 453.546,Z 55.989,A -85,B 0,C 180,E1 -8206.196,E2 -8206.196} C_VEL
LIN {X 0,Y 453.522,Z 55.989,A -85,B 0,C 180,E1 -8209.041,E2 -8209.041} C_VEL
LIN {X 0,Y 453.478,Z 55.996,A -85,B 0,C 180,E1 -8211.836,E2 -8211.836} C_VEL
LIN {X 0,Y 453.503,Z 55.992,A -85,B 0,C 180,E1 -8214.735,E2 -8214.735} C_VEL
LIN {X 0,Y 453.54,Z 55.992,A -85,B 0,C 180,E1 -8217.961,E2 -8217.961} C_VEL
LIN {X 0,Y 453.468,Z 55.997,A -85,B 0,C 180,E1 -8221.525,E2 -8221.525} C_VEL
LIN {X 0,Y 453.491,Z 55.992,A -85,B 0,C 180,E1 -8224.778,E2 -8224.778} C_VEL
LIN {X 0,Y 453.475,Z 55.995,A -85,B 0,C 180,E1 -8228.311,E2 -8228.311} C_VEL
LIN {X 0,Y 453.496,Z 55.991,A -85,B 0,C 180,E1 -8230.609,E2 -8230.609} C_VEL
LIN {X 0,Y 453.457,Z 56,A -85,B 0,C 180,E1 -8233.244,E2 -8233.244} C_VEL
LIN {X 0,Y 453.466,Z 55.999,A -85,B 0,C 180,E1 -8235.779,E2 -8235.779} C_VEL
LIN {X 0,Y 453.482,Z 55.993,A -85,B 0,C 180,E1 -8238.21,E2 -8238.21} C_VEL
LIN {X 0,Y 453.494,Z 55.994,A -85,B 0,C 180,E1 -8240.794,E2 -8240.794} C_VEL
LIN {X 0,Y 453.458,Z 55.997,A -85,B 0,C 180,E1 -8243.918,E2 -8243.918} C_VEL
LIN {X 0,Y 453.486,Z 55.999,A -85,B 0,C 180,E1 -8247.152,E2 -8247.152} C_VEL
LIN {X 0,Y 453.479,Z 55.994,A -85,B 0,C 180,E1 -8250.269,E2 -8250.269} C_VEL
LIN {X 0,Y 453.511,Z 55.992,A -85,B 0,C 180,E1 -8253.294,E2 -8253.294} C_VEL
LIN {X 0,Y 453.506,Z 55.992,A -85,B 0,C 180,E1 -8256.239,E2 -8256.239} C_VEL
LIN {X 0,Y 453.487,Z 55.994,A -85,B 0,C 180,E1 -8259.118,E2 -8259.118} C_VEL
LIN {X 0,Y 453.506,Z 55.992,A -85,B 0,C 180,E1 -8261.944,E2 -8261.944} C_VEL
LIN {X 0,Y 453.545,Z 55.989,A -85,B 0,C 180,E1 -8264.727,E2 -8264.727} C_VEL
LIN {X 0,Y 453.564,Z 55.989,A -85,B 0,C 180,E1 -8268.379,E2 -8268.379} C_VEL
LIN {X 0,Y 453.59,Z 55.98,A -85,B 0,C 180,E1 -8271.087,E2 -8271.087} C_VEL
LIN {X 0,Y 453.674,Z 55.973,A -85,B 0,C 180,E1 -8273.775,E2 -8273.775} C_VEL
LIN {X 0,Y 453.741,Z 55.962,A -85,B 0,C 180,E1 -8277.337,E2 -8277.337} C_VEL
LIN {X 0,Y 453.828,Z 55.956,A -85,B 0,C 180,E1 -8280,E2 -8280} C_VEL
LIN {X 0,Y 453.748,Z 55.96,A -85,B 0,C 180,E1 -8282.663,E2 -8282.663} C_VEL
LIN {X 0,Y 453.651,Z 55.973,A -85,B 0,C 180,E1 -8286.226,E2 -8286.226} C_VEL
LIN {X 0,Y 453.59,Z 55.981,A -85,B 0,C 180,E1 -8288.914,E2 -8288.914} C_VEL
LIN {X 0,Y 453.569,Z 55.982,A -85,B 0,C 180,E1 -8292.529,E2 -8292.529} C_VEL
LIN {X 0,Y 453.549,Z 55.985,A -85,B 0,C 180,E1 -8296.196,E2 -8296.196} C_VEL
LIN {X 0,Y 453.522,Z 55.994,A -85,B 0,C 180,E1 -8299.039,E2 -8299.039} C_VEL
LIN {X 0,Y 453.481,Z 55.994,A -85,B 0,C 180,E1 -8301.836,E2 -8301.836} C_VEL
LIN {X 0,Y 453.505,Z 55.995,A -85,B 0,C 180,E1 -8304.735,E2 -8304.735} C_VEL
LIN {X 0,Y 453.511,Z 55.99,A -85,B 0,C 180,E1 -8307.953,E2 -8307.953} C_VEL
LIN {X 0,Y 453.48,Z 56.001,A -85,B 0,C 180,E1 -8310.759,E2 -8310.759} C_VEL
LIN {X 0,Y 453.472,Z 55.995,A -85,B 0,C 180,E1 -8313.913,E2 -8313.913} C_VEL
LIN {X 0,Y 453.456,Z 55.997,A -85,B 0,C 180,E1 -8317.19,E2 -8317.19} C_VEL
LIN {X 0,Y 453.487,Z 55.992,A -85,B 0,C 180,E1 -8319.45,E2 -8319.45} C_VEL
LIN {X 0,Y 453.48,Z 55.996,A -85,B 0,C 180,E1 -8321.935,E2 -8321.935} C_VEL
LIN {X 0,Y 453.486,Z 55.993,A -85,B 0,C 180,E1 -8325.471,E2 -8325.471} C_VEL
LIN {X 0,Y 453.467,Z 56.002,A -85,B 0,C 180,E1 -8328.207,E2 -8328.207} C_VEL
LIN {X 0,Y 453.453,Z 55.997,A -85,B 0,C 180,E1 -8330.8,E2 -8330.8} C_VEL
LIN {X 0,Y 453.455,Z 56.004,A -85,B 0,C 180,E1 -8333.917,E2 -8333.917} C_VEL
LIN {X 0,Y 453.482,Z 55.994,A -85,B 0,C 180,E1 -8337.151,E2 -8337.151} C_VEL
LIN {X 0,Y 453.478,Z 55.999,A -85,B 0,C 180,E1 -8340.268,E2 -8340.268} C_VEL
LIN {X 0,Y 453.619,Z 56.161,A -85,B 0,C 180,E1 -8343.021,E2 -8343.021} C_VEL
LIN {X 0,Y 455.819,Z 67.843,A -85,B 0,C 180,E1 -8345.156,E2 -8345.156} C_VEL
LIN {X 0,Y 455.512,Z 77.673,A -85,B 0,C 180,E1 -8346.831,E2 -8346.831} C_VEL
LIN {X 0,Y 454.75,Z 95.831,A -85,B 0,C 180,E1 -8349.887,E2 -8349.887} C_VEL
LIN {X 0,Y 454.132,Z 112.19,A -85,B 0,C 180,E1 -8352.616,E2 -8352.616} C_VEL
LIN {X 0,Y 457.167,Z 136.678,A -85,B 0,C 180,E1 -8353.112,E2 -8353.112} C_VEL
LIN {X 0,Y 456.491,Z 221.092,A -85,B 0,C 180,E1 -8354.456,E2 -8354.456} C_VEL
LIN {X 0,Y 456.033,Z 234.389,A -85,B 0,C 180,E1 -8354.84,E2 -8354.84} C_VEL
LIN {X 0,Y 455.579,Z 246.604,A -85,B 0,C 180,E1 -8355.368,E2 -8355.368} C_VEL
LIN {X 0,Y 455.077,Z 258.113,A -85,B 0,C 180,E1 -8356.036,E2 -8356.036} C_VEL
LIN {X 0,Y 454.491,Z 269.875,A -85,B 0,C 180,E1 -8356.925,E2 -8356.925} C_VEL
LIN {X 0,Y 453.937,Z 280.53,A -85,B 0,C 180,E1 -8357.935,E2 -8357.935} C_VEL
LIN {X 0,Y 453.533,Z 290.088,A -85,B 0,C 180,E1 -8359.057,E2 -8359.057} C_VEL
LIN {X 0,Y 453.072,Z 299.276,A -85,B 0,C 180,E1 -8360.401,E2 -8360.401} C_VEL
LIN {X 0,Y 452.814,Z 306.683,A -85,B 0,C 180,E1 -8361.746,E2 -8361.746} C_VEL
LIN {X 0,Y 452.658,Z 311.701,A -85,B 0,C 180,E1 -8362.865,E2 -8362.865} C_VEL
LIN {X 0,Y 452.525,Z 316.947,A -85,B 0,C 180,E1 -8364.324,E2 -8364.324} C_VEL
LIN {X 0,Y 452.495,Z 320.299,A -85,B 0,C 180,E1 -8365.546,E2 -8365.546} C_VEL
LIN {X 0,Y 452.568,Z 322.229,A -85,B 0,C 180,E1 -8366.439,E2 -8366.439} C_VEL
LIN {X 0,Y 452.555,Z 323.708,A -85,B 0,C 180,E1 -8367.33,E2 -8367.33} C_VEL
LIN {X 0,Y 452.544,Z 324.745,A -85,B 0,C 180,E1 -8368.22,E2 -8368.22} C_VEL
LIN {X 0,Y 452.488,Z 325.645,A -85,B 0,C 180,E1 -8370,E2 -8370} C_VEL
LIN {X 0,Y 452.505,Z 325.492,A -85,B 0,C 180,E1 -8370.89,E2 -8370.89} C_VEL
LIN {X 0,Y 452.553,Z 323.945,A -85,B 0,C 180,E1 -8372.67,E2 -8372.67} C_VEL
LIN {X 0,Y 452.536,Z 322.578,A -85,B 0,C 180,E1 -8373.562,E2 -8373.562} C_VEL
LIN {X 0,Y 452.539,Z 319.696,A -85,B 0,C 180,E1 -8374.9,E2 -8374.9} C_VEL
LIN {X 0,Y 452.554,Z 315.493,A -85,B 0,C 180,E1 -8376.331,E2 -8376.331} C_VEL
LIN {X 0,Y 452.72,Z 310.754,A -85,B 0,C 180,E1 -8377.582,E2 -8377.582} C_VEL
LIN {X 0,Y 452.926,Z 304.447,A -85,B 0,C 180,E1 -8378.927,E2 -8378.927} C_VEL
LIN {X 0,Y 453.283,Z 296.578,A -85,B 0,C 180,E1 -8380.271,E2 -8380.271} C_VEL
LIN {X 0,Y 453.916,Z 286.791,A -85,B 0,C 180,E1 -8381.612,E2 -8381.612} C_VEL
LIN {X 0,Y 454.477,Z 276.478,A -85,B 0,C 180,E1 -8382.748,E2 -8382.748} C_VEL
LIN {X 0,Y 455.13,Z 265.223,A -85,B 0,C 180,E1 -8383.734,E2 -8383.734} C_VEL
LIN {X 0,Y 455.733,Z 254.015,A -85,B 0,C 180,E1 -8384.513,E2 -8384.513} C_VEL
LIN {X 0,Y 456.355,Z 242.677,A -85,B 0,C 180,E1 -8385.12,E2 -8385.12} C_VEL
LIN {X 0,Y 456.863,Z 230.762,A -85,B 0,C 180,E1 -8385.588,E2 -8385.588} C_VEL
LIN {X 0,Y 457.215,Z 217.803,A -85,B 0,C 180,E1 -8385.919,E2 -8385.919} C_VEL
LIN {X 0,Y 457.86,Z 134.698,A -85,B 0,C 180,E1 -8387.253,E2 -8387.253} C_VEL
LIN {X 0,Y 454.814,Z 114.421,A -85,B 0,C 180,E1 -8387.72,E2 -8387.72} C_VEL
LIN {X 0,Y 454.384,Z 111.71,A -85,B 0,C 180,E1 -8387.81,E2 -8387.81} C_VEL
LIN {X 0,Y 455.15,Z 95.52,A -85,B 0,C 180,E1 -8390.566,E2 -8390.566} C_VEL
LIN {X 0,Y 456.056,Z 77.834,A -85,B 0,C 180,E1 -8393.62,E2 -8393.62} C_VEL
LIN {X 0,Y 456.393,Z 69.668,A -85,B 0,C 180,E1 -8395.056,E2 -8395.056} C_VEL
LIN {X 0,Y 453.896,Z 57.411,A -85,B 0,C 180,E1 -8397.429,E2 -8397.429} C_VEL
LIN {X 0,Y 453.547,Z 55.992,A -85,B 0,C 180,E1 -8397.744,E2 -8397.744} C_VEL
LIN {X 0,Y 453.479,Z 55.995,A -85,B 0,C 180,E1 -8400.759,E2 -8400.759} C_VEL
LIN {X 0,Y 453.471,Z 56,A -85,B 0,C 180,E1 -8403.913,E2 -8403.913} C_VEL
LIN {X 0,Y 453.455,Z 55.998,A -85,B 0,C 180,E1 -8407.19,E2 -8407.19} C_VEL
LIN {X 0,Y 453.492,Z 55.99,A -85,B 0,C 180,E1 -8409.45,E2 -8409.45} C_VEL
LIN {X 0,Y 453.479,Z 55.997,A -85,B 0,C 180,E1 -8411.935,E2 -8411.935} C_VEL
LIN {X 0,Y 453.487,Z 55.995,A -85,B 0,C 180,E1 -8415.471,E2 -8415.471} C_VEL
LIN {X 0,Y 453.482,Z 55.993,A -85,B 0,C 180,E1 -8418.209,E2 -8418.209} C_VEL
LIN {X 0,Y 453.49,Z 55.99,A -85,B 0,C 180,E1 -8420.794,E2 -8420.794} C_VEL
LIN {X 0,Y 453.457,Z 55.997,A -85,B 0,C 180,E1 -8423.917,E2 -8423.917} C_VEL
LIN {X 0,Y 453.482,Z 55.996,A -85,B 0,C 180,E1 -8427.151,E2 -8427.151} C_VEL
LIN {X 0,Y 453.479,Z 55.991,A -85,B 0,C 180,E1 -8430.268,E2 -8430.268} C_VEL
LIN {X 0,Y 453.508,Z 55.99,A -85,B 0,C 180,E1 -8433.294,E2 -8433.294} C_VEL
LIN {X 0,Y 453.505,Z 55.993,A -85,B 0,C 180,E1 -8436.239,E2 -8436.239} C_VEL
LIN {X 0,Y 453.487,Z 55.995,A -85,B 0,C 180,E1 -8439.118,E2 -8439.118} C_VEL
LIN {X 0,Y 453.514,Z 55.99,A -85,B 0,C 180,E1 -8441.945,E2 -8441.945} C_VEL
LIN {X 0,Y 453.544,Z 55.99,A -85,B 0,C 180,E1 -8444.726,E2 -8444.726} C_VEL
LIN {X 0,Y 453.564,Z 55.985,A -85,B 0,C 180,E1 -8448.379,E2 -8448.379} C_VEL
LIN {X 0,Y 453.656,Z 55.976,A -85,B 0,C 180,E1 -8451.985,E2 -8451.985} C_VEL
LIN {X 0,Y 453.672,Z 55.971,A -85,B 0,C 180,E1 -8454.667,E2 -8454.667} C_VEL
LIN {X 0,Y 453.741,Z 55.962,A -85,B 0,C 180,E1 -8457.337,E2 -8457.337} C_VEL
LIN {X 0,Y 453.827,Z 55.956,A -85,B 0,C 180,E1 -8460,E2 -8460} C_VEL
LIN {X 0,Y 453.747,Z 55.958,A -85,B 0,C 180,E1 -8462.663,E2 -8462.663} C_VEL
LIN {X 0,Y 453.663,Z 55.972,A -85,B 0,C 180,E1 -8466.225,E2 -8466.225} C_VEL
LIN {X 0,Y 453.589,Z 55.978,A -85,B 0,C 180,E1 -8468.913,E2 -8468.913} C_VEL
LIN {X 0,Y 453.567,Z 55.983,A -85,B 0,C 180,E1 -8472.529,E2 -8472.529} C_VEL
LIN {X 0,Y 453.548,Z 55.986,A -85,B 0,C 180,E1 -8476.196,E2 -8476.196} C_VEL
LIN {X 0,Y 453.52,Z 55.991,A -85,B 0,C 180,E1 -8479.039,E2 -8479.039} C_VEL
LIN {X 0,Y 453.48,Z 55.993,A -85,B 0,C 180,E1 -8481.836,E2 -8481.836} C_VEL
LIN {X 0,Y 453.508,Z 55.996,A -85,B 0,C 180,E1 -8484.735,E2 -8484.735} C_VEL
LIN {X 0,Y 453.509,Z 55.989,A -85,B 0,C 180,E1 -8487.953,E2 -8487.953} C_VEL
LIN {X 0,Y 453.478,Z 55.997,A -85,B 0,C 180,E1 -8490.759,E2 -8490.759} C_VEL
LIN {X 0,Y 453.47,Z 55.996,A -85,B 0,C 180,E1 -8493.913,E2 -8493.913} C_VEL
LIN {X 0,Y 453.451,Z 55.997,A -85,B 0,C 180,E1 -8497.19,E2 -8497.19} C_VEL
LIN {X 0,Y 453.495,Z 55.987,A -85,B 0,C 180,E1 -8500.609,E2 -8500.609} C_VEL
LIN {X 0,Y 453.462,Z 56.002,A -85,B 0,C 180,E1 -8504.222,E2 -8504.222} C_VEL
LIN {X 0,Y 453.449,Z 56,A -85,B 0,C 180,E1 -8507.003,E2 -8507.003} C_VEL
LIN {X 0,Y 453.495,Z 55.997,A -85,B 0,C 180,E1 -8509.409,E2 -8509.409} C_VEL
LIN {X 0,Y 453.45,Z 56.001,A -85,B 0,C 180,E1 -8512.81,E2 -8512.81} C_VEL
LIN {X 0,Y 453.469,Z 56.001,A -85,B 0,C 180,E1 -8516.086,E2 -8516.086} C_VEL
LIN {X 0,Y 453.483,Z 56.004,A -85,B 0,C 180,E1 -8519.612,E2 -8519.612} C_VEL
LIN {X 0,Y 453.497,Z 56.16,A -85,B 0,C 180,E1 -8519.736,E2 -8519.736} C_VEL
LIN {X 0,Y 454.956,Z 64.309,A -85,B 0,C 180,E1 -8521.705,E2 -8521.705} C_VEL
LIN {X 0,Y 455.024,Z 67.18,A -85,B 0,C 180,E1 -8522.305,E2 -8522.305} C_VEL
LIN {X 0,Y 458.39,Z 81.483,A -85,B 0,C 180,E1 -8522.696,E2 -8522.696} C_VEL
LIN {X 0,Y 457.431,Z 173.739,A -85,B 0,C 180,E1 -8524.184,E2 -8524.184} C_VEL
LIN {X 0,Y 457.211,Z 187.048,A -85,B 0,C 180,E1 -8524.588,E2 -8524.588} C_VEL
LIN {X 0,Y 456.866,Z 199.253,A -85,B 0,C 180,E1 -8525.133,E2 -8525.133} C_VEL
LIN {X 0,Y 456.311,Z 211.34,A -85,B 0,C 180,E1 -8525.863,E2 -8525.863} C_VEL
LIN {X 0,Y 455.391,Z 216.549,A -85,B 0,C 180,E1 -8526.217,E2 -8526.217} C_VEL
LIN {X 0,Y 452.187,Z 224.756,A -85,B 0,C 180,E1 -8526.797,E2 -8526.797} C_VEL
LIN {X 0,Y 448.987,Z 232.464,A -85,B 0,C 180,E1 -8527.462,E2 -8527.462} C_VEL
LIN {X 0,Y 448.071,Z 236.852,A -85,B 0,C 180,E1 -8527.941,E2 -8527.941} C_VEL
LIN {X 0,Y 447.486,Z 245.388,A -85,B 0,C 180,E1 -8529.065,E2 -8529.065} C_VEL
LIN {X 0,Y 446.993,Z 253.004,A -85,B 0,C 180,E1 -8530.29,E2 -8530.29} C_VEL
LIN {X 0,Y 446.5,Z 259.853,A -85,B 0,C 180,E1 -8531.651,E2 -8531.651} C_VEL
LIN {X 0,Y 446.132,Z 265.487,A -85,B 0,C 180,E1 -8533.056,E2 -8533.056} C_VEL
LIN {X 0,Y 445.858,Z 269.866,A -85,B 0,C 180,E1 -8534.457,E2 -8534.457} C_VEL
LIN {X 0,Y 445.727,Z 272.167,A -85,B 0,C 180,E1 -8535.387,E2 -8535.387} C_VEL
LIN {X 0,Y 445.6,Z 274.004,A -85,B 0,C 180,E1 -8536.315,E2 -8536.315} C_VEL
LIN {X 0,Y 445.495,Z 276.166,A -85,B 0,C 180,E1 -8537.985,E2 -8537.985} C_VEL
LIN {X 0,Y 445.462,Z 276.884,A -85,B 0,C 180,E1 -8539.087,E2 -8539.087} C_VEL
LIN {X 0,Y 445.396,Z 277.018,A -85,B 0,C 180,E1 -8540.004,E2 -8540.004} C_VEL
LIN {X 0,Y 445.47,Z 276.074,A -85,B 0,C 180,E1 -8541.837,E2 -8541.837} C_VEL
LIN {X 0,Y 445.617,Z 273.806,A -85,B 0,C 180,E1 -8543.513,E2 -8543.513} C_VEL
LIN {X 0,Y 445.668,Z 270.502,A -85,B 0,C 180,E1 -8545.024,E2 -8545.024} C_VEL
LIN {X 0,Y 445.911,Z 266.428,A -85,B 0,C 180,E1 -8546.386,E2 -8546.386} C_VEL
LIN {X 0,Y 446.075,Z 261.218,A -85,B 0,C 180,E1 -8547.743,E2 -8547.743} C_VEL
LIN {X 0,Y 446.488,Z 254.668,A -85,B 0,C 180,E1 -8549.098,E2 -8549.098} C_VEL
LIN {X 0,Y 446.91,Z 246.56,A -85,B 0,C 180,E1 -8550.451,E2 -8550.451} C_VEL
LIN {X 0,Y 447.289,Z 238.289,A -85,B 0,C 180,E1 -8551.576,E2 -8551.576} C_VEL
LIN {X 0,Y 447.875,Z 229.221,A -85,B 0,C 180,E1 -8552.586,E2 -8552.586} C_VEL
LIN {X 0,Y 448.428,Z 219.374,A -85,B 0,C 180,E1 -8553.482,E2 -8553.482} C_VEL
LIN {X 0,Y 448.944,Z 208.696,A -85,B 0,C 180,E1 -8554.264,E2 -8554.264} C_VEL
LIN {X 0,Y 449.303,Z 197.006,A -85,B 0,C 180,E1 -8554.935,E2 -8554.935} C_VEL
LIN {X 0,Y 449.582,Z 184.436,A -85,B 0,C 180,E1 -8555.466,E2 -8555.466} C_VEL
LIN {X 0,Y 449.835,Z 172.332,A -85,B 0,C 180,E1 -8555.801,E2 -8555.801} C_VEL
LIN {X 0,Y 450.542,Z 81.543,A -85,B 0,C 180,E1 -8557.264,E2 -8557.264} C_VEL
LIN {X 0,Y 447.678,Z 66.888,A -85,B 0,C 180,E1 -8557.612,E2 -8557.612} C_VEL
LIN {X 0,Y 447.396,Z 61.964,A -85,B 0,C 180,E1 -8558.729,E2 -8558.729} C_VEL
LIN {X 0,Y 446.523,Z 56.867,A -85,B 0,C 180,E1 -8559.97,E2 -8559.97} C_VEL
LIN {X 0,Y 446.523,Z 56.867,A -85,B 0,C 180,E1 -8562.73,E2 -8562.73} C_VEL
LIN {X 0,Y 446.498,Z 56.867,A -85,B 0,C 180,E1 -8566.228,E2 -8566.228} C_VEL
LIN {X 0,Y 446.471,Z 56.867,A -85,B 0,C 180,E1 -8569.303,E2 -8569.303} C_VEL
LIN {X 0,Y 446.42,Z 56.879,A -85,B 0,C 180,E1 -8572.2,E2 -8572.2} C_VEL
LIN {X 0,Y 446.446,Z 56.87,A -85,B 0,C 180,E1 -8575.153,E2 -8575.153} C_VEL
LIN {X 0,Y 446.486,Z 56.871,A -85,B 0,C 180,E1 -8578.179,E2 -8578.179} C_VEL
LIN {X 0,Y 446.421,Z 56.878,A -85,B 0,C 180,E1 -8581.775,E2 -8581.775} C_VEL
LIN {X 0,Y 446.432,Z 56.872,A -85,B 0,C 180,E1 -8584.523,E2 -8584.523} C_VEL
LIN {X 0,Y 446.433,Z 56.874,A -85,B 0,C 180,E1 -8588.082,E2 -8588.082} C_VEL
LIN {X 0,Y 446.429,Z 56.872,A -85,B 0,C 180,E1 -8590.918,E2 -8590.918} C_VEL
LIN {X 0,Y 446.403,Z 56.879,A -85,B 0,C 180,E1 -8593.846,E2 -8593.846} C_VEL
LIN {X 0,Y 446.4,Z 56.875,A -85,B 0,C 180,E1 -8596.404,E2 -8596.404} C_VEL
LIN {X 0,Y 446.429,Z 56.876,A -85,B 0,C 180,E1 -8599.083,E2 -8599.083} C_VEL
LIN {X 0,Y 446.412,Z 56.874,A -85,B 0,C 180,E1 -8602.122,E2 -8602.122} C_VEL
LIN {X 0,Y 446.433,Z 56.874,A -85,B 0,C 180,E1 -8605.477,E2 -8605.477} C_VEL
LIN {X 0,Y 446.42,Z 56.877,A -85,B 0,C 180,E1 -8608.7,E2 -8608.7} C_VEL
LIN {X 0,Y 446.488,Z 56.864,A -85,B 0,C 180,E1 -8611.822,E2 -8611.822} C_VEL
LIN {X 0,Y 446.462,Z 56.874,A -85,B 0,C 180,E1 -8614.848,E2 -8614.848} C_VEL
LIN {X 0,Y 446.453,Z 56.872,A -85,B 0,C 180,E1 -8618.245,E2 -8618.245} C_VEL
LIN {X 0,Y 446.455,Z 56.869,A -85,B 0,C 180,E1 -8621.649,E2 -8621.649} C_VEL
LIN {X 0,Y 446.513,Z 56.868,A -85,B 0,C 180,E1 -8624.48,E2 -8624.48} C_VEL
LIN {X 0,Y 446.522,Z 56.867,A -85,B 0,C 180,E1 -8628.193,E2 -8628.193} C_VEL
LIN {X 0,Y 446.537,Z 56.859,A -85,B 0,C 180,E1 -8630.945,E2 -8630.945} C_VEL
LIN {X 0,Y 446.642,Z 56.848,A -85,B 0,C 180,E1 -8633.676,E2 -8633.676} C_VEL
LIN {X 0,Y 446.688,Z 56.84,A -85,B 0,C 180,E1 -8637.295,E2 -8637.295} C_VEL
LIN {X 0,Y 446.798,Z 56.831,A -85,B 0,C 180,E1 -8640,E2 -8640} C_VEL
LIN {X 0,Y 446.695,Z 56.839,A -85,B 0,C 180,E1 -8642.705,E2 -8642.705} C_VEL
LIN {X 0,Y 446.62,Z 56.849,A -85,B 0,C 180,E1 -8646.324,E2 -8646.324} C_VEL
LIN {X 0,Y 446.537,Z 56.86,A -85,B 0,C 180,E1 -8649.055,E2 -8649.055} C_VEL
LIN {X 0,Y 446.527,Z 56.86,A -85,B 0,C 180,E1 -8652.73,E2 -8652.73} C_VEL
LIN {X 0,Y 446.501,Z 56.863,A -85,B 0,C 180,E1 -8656.227,E2 -8656.227} C_VEL
LIN {X 0,Y 446.473,Z 56.872,A -85,B 0,C 180,E1 -8659.303,E2 -8659.303} C_VEL
LIN {X 0,Y 446.423,Z 56.873,A -85,B 0,C 180,E1 -8662.2,E2 -8662.2} C_VEL
LIN {X 0,Y 446.447,Z 56.874,A -85,B 0,C 180,E1 -8665.153,E2 -8665.153} C_VEL
LIN {X 0,Y 446.454,Z 56.87,A -85,B 0,C 180,E1 -8668.181,E2 -8668.181} C_VEL
LIN {X 0,Y 446.42,Z 56.874,A -85,B 0,C 180,E1 -8671.3,E2 -8671.3} C_VEL
LIN {X 0,Y 446.427,Z 56.879,A -85,B 0,C 180,E1 -8674.523,E2 -8674.523} C_VEL
LIN {X 0,Y 446.417,Z 56.876,A -85,B 0,C 180,E1 -8678.079,E2 -8678.079} C_VEL
LIN {X 0,Y 446.43,Z 56.873,A -85,B 0,C 180,E1 -8680.917,E2 -8680.917} C_VEL
LIN {X 0,Y 446.402,Z 56.878,A -85,B 0,C 180,E1 -8683.846,E2 -8683.846} C_VEL
LIN {X 0,Y 446.401,Z 56.88,A -85,B 0,C 180,E1 -8686.403,E2 -8686.403} C_VEL
LIN {X 0,Y 446.435,Z 56.875,A -85,B 0,C 180,E1 -8689.801,E2 -8689.801} C_VEL
LIN {X 0,Y 446.403,Z 56.876,A -85,B 0,C 180,E1 -8693.254,E2 -8693.254} C_VEL
LIN {X 0,Y 446.451,Z 56.869,A -85,B 0,C 180,E1 -8696.566,E2 -8696.566} C_VEL
LIN {X 0,Y 446.434,Z 56.879,A -85,B 0,C 180,E1 -8699.979,E2 -8699.979} C_VEL
LIN {X 0,Y 446.555,Z 56.937,A -85,B 0,C 180,E1 -8702.812,E2 -8702.812} C_VEL
LIN {X 0,Y 448.942,Z 69.955,A -85,B 0,C 180,E1 -8705.226,E2 -8705.226} C_VEL
LIN {X 0,Y 448.121,Z 88.258,A -85,B 0,C 180,E1 -8708.373,E2 -8708.373} C_VEL
LIN {X 0,Y 447.27,Z 107.744,A -85,B 0,C 180,E1 -8711.683,E2 -8711.683} C_VEL
LIN {X 0,Y 447.104,Z 111.828,A -85,B 0,C 180,E1 -8712.374,E2 -8712.374} C_VEL
LIN {X 0,Y 450.308,Z 137.238,A -85,B 0,C 180,E1 -8712.897,E2 -8712.897} C_VEL
LIN {X 0,Y 449.596,Z 220.524,A -85,B 0,C 180,E1 -8714.24,E2 -8714.24} C_VEL
LIN {X 0,Y 449.124,Z 233.889,A -85,B 0,C 180,E1 -8714.63,E2 -8714.63} C_VEL
LIN {X 0,Y 448.635,Z 246.709,A -85,B 0,C 180,E1 -8715.194,E2 -8715.194} C_VEL
LIN {X 0,Y 448.058,Z 258.885,A -85,B 0,C 180,E1 -8715.929,E2 -8715.929} C_VEL
LIN {X 0,Y 447.425,Z 270.937,A -85,B 0,C 180,E1 -8716.875,E2 -8716.875} C_VEL
LIN {X 0,Y 446.883,Z 280.923,A -85,B 0,C 180,E1 -8717.857,E2 -8717.857} C_VEL
LIN {X 0,Y 446.504,Z 289.465,A -85,B 0,C 180,E1 -8718.883,E2 -8718.883} C_VEL
LIN {X 0,Y 446.001,Z 298.704,A -85,B 0,C 180,E1 -8720.247,E2 -8720.247} C_VEL
LIN {X 0,Y 445.753,Z 306.149,A -85,B 0,C 180,E1 -8721.614,E2 -8721.614} C_VEL
LIN {X 0,Y 445.51,Z 312.974,A -85,B 0,C 180,E1 -8723.205,E2 -8723.205} C_VEL
LIN {X 0,Y 445.466,Z 317.476,A -85,B 0,C 180,E1 -8724.568,E2 -8724.568} C_VEL
LIN {X 0,Y 445.419,Z 319.846,A -85,B 0,C 180,E1 -8725.475,E2 -8725.475} C_VEL
LIN {X 0,Y 445.465,Z 321.786,A -85,B 0,C 180,E1 -8726.382,E2 -8726.382} C_VEL
LIN {X 0,Y 445.48,Z 323.288,A -85,B 0,C 180,E1 -8727.287,E2 -8727.287} C_VEL
LIN {X 0,Y 445.456,Z 324.336,A -85,B 0,C 180,E1 -8728.192,E2 -8728.192} C_VEL
LIN {X 0,Y 445.442,Z 324.991,A -85,B 0,C 180,E1 -8729.096,E2 -8729.096} C_VEL
LIN {X 0,Y 445.422,Z 325.256,A -85,B 0,C 180,E1 -8730,E2 -8730} C_VEL
LIN {X 0,Y 445.441,Z 325.122,A -85,B 0,C 180,E1 -8730.904,E2 -8730.904} C_VEL
LIN {X 0,Y 445.476,Z 323.596,A -85,B 0,C 180,E1 -8732.713,E2 -8732.713} C_VEL
LIN {X 0,Y 445.433,Z 322.238,A -85,B 0,C 180,E1 -8733.618,E2 -8733.618} C_VEL
LIN {X 0,Y 445.465,Z 319.378,A -85,B 0,C 180,E1 -8734.978,E2 -8734.978} C_VEL
LIN {X 0,Y 445.455,Z 315.49,A -85,B 0,C 180,E1 -8736.341,E2 -8736.341} C_VEL
LIN {X 0,Y 445.67,Z 310.487,A -85,B 0,C 180,E1 -8737.703,E2 -8737.703} C_VEL
LIN {X 0,Y 445.892,Z 304.211,A -85,B 0,C 180,E1 -8739.069,E2 -8739.069} C_VEL
LIN {X 0,Y 446.27,Z 296.395,A -85,B 0,C 180,E1 -8740.434,E2 -8740.434} C_VEL
LIN {X 0,Y 446.939,Z 286.652,A -85,B 0,C 180,E1 -8741.796,E2 -8741.796} C_VEL
LIN {X 0,Y 447.496,Z 277.187,A -85,B 0,C 180,E1 -8742.871,E2 -8742.871} C_VEL
LIN {X 0,Y 448.126,Z 266.674,A -85,B 0,C 180,E1 -8743.837,E2 -8743.837} C_VEL
LIN {X 0,Y 448.876,Z 254.147,A -85,B 0,C 180,E1 -8744.74,E2 -8744.74} C_VEL
LIN {X 0,Y 449.542,Z 241.819,A -85,B 0,C 180,E1 -8745.413,E2 -8745.413} C_VEL
LIN {X 0,Y 450.13,Z 229.648,A -85,B 0,C 180,E1 -8745.886,E2 -8745.886} C_VEL
LIN {X 0,Y 450.474,Z 216.232,A -85,B 0,C 180,E1 -8746.222,E2 -8746.222} C_VEL
LIN {X 0,Y 451.124,Z 135.289,A -85,B 0,C 180,E1 -8747.539,E2 -8747.539} C_VEL
LIN {X 0,Y 447.89,Z 114.019,A -85,B 0,C 180,E1 -8748.042,E2 -8748.042} C_VEL
LIN {X 0,Y 447.465,Z 111.469,A -85,B 0,C 180,E1 -8748.106,E2 -8748.106} C_VEL
LIN {X 0,Y 448.23,Z 95.36,A -85,B 0,C 180,E1 -8750.898,E2 -8750.898} C_VEL
LIN {X 0,Y 449.063,Z 80.424,A -85,B 0,C 180,E1 -8753.521,E2 -8753.521} C_VEL
LIN {X 0,Y 449.553,Z 72.276,A -85,B 0,C 180,E1 -8754.967,E2 -8754.967} C_VEL
LIN {X 0,Y 448.062,Z 63.797,A -85,B 0,C 180,E1 -8756.611,E2 -8756.611} C_VEL
LIN {X 0,Y 446.49,Z 56.871,A -85,B 0,C 180,E1 -8758.006,E2 -8758.006} C_VEL
LIN {X 0,Y 446.418,Z 56.874,A -85,B 0,C 180,E1 -8761.3,E2 -8761.3} C_VEL
LIN {X 0,Y 446.426,Z 56.877,A -85,B 0,C 180,E1 -8764.524,E2 -8764.524} C_VEL
LIN {X 0,Y 446.419,Z 56.877,A -85,B 0,C 180,E1 -8768.079,E2 -8768.079} C_VEL
LIN {X 0,Y 446.43,Z 56.872,A -85,B 0,C 180,E1 -8770.918,E2 -8770.918} C_VEL
LIN {X 0,Y 446.403,Z 56.878,A -85,B 0,C 180,E1 -8773.846,E2 -8773.846} C_VEL
LIN {X 0,Y 446.401,Z 56.874,A -85,B 0,C 180,E1 -8776.404,E2 -8776.404} C_VEL
LIN {X 0,Y 446.43,Z 56.873,A -85,B 0,C 180,E1 -8779.082,E2 -8779.082} C_VEL
LIN {X 0,Y 446.411,Z 56.873,A -85,B 0,C 180,E1 -8782.121,E2 -8782.121} C_VEL
LIN {X 0,Y 446.426,Z 56.874,A -85,B 0,C 180,E1 -8785.477,E2 -8785.477} C_VEL
LIN {X 0,Y 446.419,Z 56.877,A -85,B 0,C 180,E1 -8788.7,E2 -8788.7} C_VEL
LIN {X 0,Y 446.488,Z 56.866,A -85,B 0,C 180,E1 -8791.821,E2 -8791.821} C_VEL
LIN {X 0,Y 446.453,Z 56.872,A -85,B 0,C 180,E1 -8794.847,E2 -8794.847} C_VEL
LIN {X 0,Y 446.452,Z 56.869,A -85,B 0,C 180,E1 -8798.245,E2 -8798.245} C_VEL
LIN {X 0,Y 446.46,Z 56.868,A -85,B 0,C 180,E1 -8801.649,E2 -8801.649} C_VEL
LIN {X 0,Y 446.512,Z 56.866,A -85,B 0,C 180,E1 -8804.48,E2 -8804.48} C_VEL
LIN {X 0,Y 446.522,Z 56.86,A -85,B 0,C 180,E1 -8808.193,E2 -8808.193} C_VEL
LIN {X 0,Y 446.604,Z 56.854,A -85,B 0,C 180,E1 -8811.858,E2 -8811.858} C_VEL
LIN {X 0,Y 446.647,Z 56.847,A -85,B 0,C 180,E1 -8814.583,E2 -8814.583} C_VEL
LIN {X 0,Y 446.667,Z 56.841,A -85,B 0,C 180,E1 -8818.197,E2 -8818.197} C_VEL
LIN {X 0,Y 446.797,Z 56.832,A -85,B 0,C 180,E1 -8820,E2 -8820} C_VEL
LIN {X 0,Y 446.693,Z 56.837,A -85,B 0,C 180,E1 -8822.705,E2 -8822.705} C_VEL
LIN {X 0,Y 446.633,Z 56.848,A -85,B 0,C 180,E1 -8826.324,E2 -8826.324} C_VEL
LIN {X 0,Y 446.536,Z 56.857,A -85,B 0,C 180,E1 -8829.055,E2 -8829.055} C_VEL
LIN {X 0,Y 446.525,Z 56.861,A -85,B 0,C 180,E1 -8832.73,E2 -8832.73} C_VEL
LIN {X 0,Y 446.499,Z 56.864,A -85,B 0,C 180,E1 -8836.227,E2 -8836.227} C_VEL
LIN {X 0,Y 446.471,Z 56.87,A -85,B 0,C 180,E1 -8839.303,E2 -8839.303} C_VEL
LIN {X 0,Y 446.421,Z 56.873,A -85,B 0,C 180,E1 -8842.199,E2 -8842.199} C_VEL
LIN {X 0,Y 446.448,Z 56.873,A -85,B 0,C 180,E1 -8845.153,E2 -8845.153} C_VEL
LIN {X 0,Y 446.452,Z 56.87,A -85,B 0,C 180,E1 -8848.181,E2 -8848.181} C_VEL
LIN {X 0,Y 446.418,Z 56.874,A -85,B 0,C 180,E1 -8851.3,E2 -8851.3} C_VEL
LIN {X 0,Y 446.425,Z 56.877,A -85,B 0,C 180,E1 -8854.523,E2 -8854.523} C_VEL
LIN {X 0,Y 446.413,Z 56.879,A -85,B 0,C 180,E1 -8858.078,E2 -8858.078} C_VEL
LIN {X 0,Y 446.42,Z 56.867,A -85,B 0,C 180,E1 -8861.392,E2 -8861.392} C_VEL
LIN {X 0,Y 446.451,Z 56.872,A -85,B 0,C 180,E1 -8865.104,E2 -8865.104} C_VEL
LIN {X 0,Y 446.42,Z 56.876,A -85,B 0,C 180,E1 -8868.608,E2 -8868.608} C_VEL
LIN {X 0,Y 446.411,Z 56.88,A -85,B 0,C 180,E1 -8871.921,E2 -8871.921} C_VEL
LIN {X 0,Y 446.424,Z 56.88,A -85,B 0,C 180,E1 -8875.476,E2 -8875.476} C_VEL
LIN {X 0,Y 446.418,Z 56.883,A -85,B 0,C 180,E1 -8878.7,E2 -8878.7} C_VEL
LIN {X 0,Y 446.46,Z 57.061,A -85,B 0,C 180,E1 -8879.491,E2 -8879.491} C_VEL
LIN {X 0,Y 448.006,Z 65.082,A -85,B 0,C 180,E1 -8881.46,E2 -8881.46} C_VEL
LIN {X 0,Y 448.098,Z 67.354,A -85,B 0,C 180,E1 -8881.977,E2 -8881.977} C_VEL
LIN {X 0,Y 451.786,Z 82.761,A -85,B 0,C 180,E1 -8882.412,E2 -8882.412} C_VEL
LIN {X 0,Y 450.71,Z 173.707,A -85,B 0,C 180,E1 -8883.895,E2 -8883.895} C_VEL
LIN {X 0,Y 450.461,Z 187.425,A -85,B 0,C 180,E1 -8884.314,E2 -8884.314} C_VEL
LIN {X 0,Y 450.071,Z 200.555,A -85,B 0,C 180,E1 -8884.916,E2 -8884.916} C_VEL
LIN {X 0,Y 449.486,Z 212.233,A -85,B 0,C 180,E1 -8885.645,E2 -8885.645} C_VEL
LIN {X 0,Y 448.813,Z 223.948,A -85,B 0,C 180,E1 -8886.587,E2 -8886.587} C_VEL
LIN {X 0,Y 448.256,Z 233.476,A -85,B 0,C 180,E1 -8887.546,E2 -8887.546} C_VEL
LIN {X 0,Y 448.071,Z 236.852,A -85,B 0,C 180,E1 -8887.941,E2 -8887.941} C_VEL
LIN {X 0,Y 447.147,Z 241.13,A -85,B 0,C 180,E1 -8888.451,E2 -8888.451} C_VEL
LIN {X 0,Y 443.89,Z 247.819,A -85,B 0,C 180,E1 -8889.296,E2 -8889.296} C_VEL
LIN {X 0,Y 440.623,Z 253.911,A -85,B 0,C 180,E1 -8890.217,E2 -8890.217} C_VEL
LIN {X 0,Y 439.697,Z 257.246,A -85,B 0,C 180,E1 -8890.84,E2 -8890.84} C_VEL
LIN {X 0,Y 439.28,Z 263.64,A -85,B 0,C 180,E1 -8892.303,E2 -8892.303} C_VEL
LIN {X 0,Y 438.921,Z 269.021,A -85,B 0,C 180,E1 -8893.888,E2 -8893.888} C_VEL
LIN {X 0,Y 438.703,Z 272.258,A -85,B 0,C 180,E1 -8895.148,E2 -8895.148} C_VEL
LIN {X 0,Y 438.554,Z 274.165,A -85,B 0,C 180,E1 -8896.091,E2 -8896.091} C_VEL
LIN {X 0,Y 438.473,Z 275.596,A -85,B 0,C 180,E1 -8897.033,E2 -8897.033} C_VEL
LIN {X 0,Y 438.422,Z 276.597,A -85,B 0,C 180,E1 -8897.972,E2 -8897.972} C_VEL
LIN {X 0,Y 438.375,Z 277.204,A -85,B 0,C 180,E1 -8898.908,E2 -8898.908} C_VEL
LIN {X 0,Y 438.325,Z 277.418,A -85,B 0,C 180,E1 -8899.842,E2 -8899.842} C_VEL
LIN {X 0,Y 438.331,Z 277.191,A -85,B 0,C 180,E1 -8900.774,E2 -8900.774} C_VEL
LIN {X 0,Y 438.457,Z 275.561,A -85,B 0,C 180,E1 -8902.633,E2 -8902.633} C_VEL
LIN {X 0,Y 438.544,Z 274.147,A -85,B 0,C 180,E1 -8903.559,E2 -8903.559} C_VEL
LIN {X 0,Y 438.589,Z 271.216,A -85,B 0,C 180,E1 -8904.944,E2 -8904.944} C_VEL
LIN {X 0,Y 438.828,Z 267.241,A -85,B 0,C 180,E1 -8906.327,E2 -8906.327} C_VEL
LIN {X 0,Y 439.009,Z 262.145,A -85,B 0,C 180,E1 -8907.706,E2 -8907.706} C_VEL
LIN {X 0,Y 439.391,Z 255.721,A -85,B 0,C 180,E1 -8909.084,E2 -8909.084} C_VEL
LIN {X 0,Y 439.841,Z 247.748,A -85,B 0,C 180,E1 -8910.458,E2 -8910.458} C_VEL
LIN {X 0,Y 440.238,Z 239.633,A -85,B 0,C 180,E1 -8911.601,E2 -8911.601} C_VEL
LIN {X 0,Y 440.852,Z 230.767,A -85,B 0,C 180,E1 -8912.627,E2 -8912.627} C_VEL
LIN {X 0,Y 441.383,Z 221.22,A -85,B 0,C 180,E1 -8913.538,E2 -8913.538} C_VEL
LIN {X 0,Y 441.934,Z 210.942,A -85,B 0,C 180,E1 -8914.332,E2 -8914.332} C_VEL
LIN {X 0,Y 442.366,Z 198.68,A -85,B 0,C 180,E1 -8915.07,E2 -8915.07} C_VEL
LIN {X 0,Y 442.664,Z 185.814,A -85,B 0,C 180,E1 -8915.638,E2 -8915.638} C_VEL
LIN {X 0,Y 442.943,Z 173.172,A -85,B 0,C 180,E1 -8916.005,E2 -8916.005} C_VEL
LIN {X 0,Y 443.783,Z 83.037,A -85,B 0,C 180,E1 -8917.479,E2 -8917.479} C_VEL
LIN {X 0,Y 440.716,Z 67.161,A -85,B 0,C 180,E1 -8917.877,E2 -8917.877} C_VEL
LIN {X 0,Y 440.153,Z 61.503,A -85,B 0,C 180,E1 -8919.188,E2 -8919.188} C_VEL
LIN {X 0,Y 439.463,Z 57.747,A -85,B 0,C 180,E1 -8920.132,E2 -8920.132} C_VEL
LIN {X 0,Y 439.467,Z 57.745,A -85,B 0,C 180,E1 -8922.938,E2 -8922.938} C_VEL
LIN {X 0,Y 439.449,Z 57.747,A -85,B 0,C 180,E1 -8926.349,E2 -8926.349} C_VEL
LIN {X 0,Y 439.404,Z 57.747,A -85,B 0,C 180,E1 -8929.626,E2 -8929.626} C_VEL
LIN {X 0,Y 439.366,Z 57.755,A -85,B 0,C 180,E1 -8932.576,E2 -8932.576} C_VEL
LIN {X 0,Y 439.399,Z 57.749,A -85,B 0,C 180,E1 -8935.586,E2 -8935.586} C_VEL
LIN {X 0,Y 439.419,Z 57.746,A -85,B 0,C 180,E1 -8938.674,E2 -8938.674} C_VEL
LIN {X 0,Y 439.372,Z 57.757,A -85,B 0,C 180,E1 -8942.031,E2 -8942.031} C_VEL
LIN {X 0,Y 439.398,Z 57.75,A -85,B 0,C 180,E1 -8945.341,E2 -8945.341} C_VEL
LIN {X 0,Y 439.393,Z 57.748,A -85,B 0,C 180,E1 -8948.594,E2 -8948.594} C_VEL
LIN {X 0,Y 439.391,Z 57.752,A -85,B 0,C 180,E1 -8951.257,E2 -8951.257} C_VEL
LIN {X 0,Y 439.402,Z 57.748,A -85,B 0,C 180,E1 -8954.73,E2 -8954.73} C_VEL
LIN {X 0,Y 439.398,Z 57.75,A -85,B 0,C 180,E1 -8957.796,E2 -8957.796} C_VEL
LIN {X 0,Y 439.413,Z 57.746,A -85,B 0,C 180,E1 -8960.226,E2 -8960.226} C_VEL
LIN {X 0,Y 439.377,Z 57.752,A -85,B 0,C 180,E1 -8963.713,E2 -8963.713} C_VEL
LIN {X 0,Y 439.377,Z 57.758,A -85,B 0,C 180,E1 -8967.054,E2 -8967.054} C_VEL
LIN {X 0,Y 439.386,Z 57.75,A -85,B 0,C 180,E1 -8970.274,E2 -8970.274} C_VEL
LIN {X 0,Y 439.432,Z 57.745,A -85,B 0,C 180,E1 -8973.397,E2 -8973.397} C_VEL
LIN {X 0,Y 439.391,Z 57.753,A -85,B 0,C 180,E1 -8976.43,E2 -8976.43} C_VEL
LIN {X 0,Y 439.392,Z 57.749,A -85,B 0,C 180,E1 -8979.397,E2 -8979.397} C_VEL
LIN {X 0,Y 439.429,Z 57.749,A -85,B 0,C 180,E1 -8982.31,E2 -8982.31} C_VEL
LIN {X 0,Y 439.452,Z 57.741,A -85,B 0,C 180,E1 -8985.174,E2 -8985.174} C_VEL
LIN {X 0,Y 439.488,Z 57.74,A -85,B 0,C 180,E1 -8988.002,E2 -8988.002} C_VEL
LIN {X 0,Y 439.536,Z 57.733,A -85,B 0,C 180,E1 -8991.726,E2 -8991.726} C_VEL
LIN {X 0,Y 439.622,Z 57.722,A -85,B 0,C 180,E1 -8994.496,E2 -8994.496} C_VEL
LIN {X 0,Y 439.638,Z 57.722,A -85,B 0,C 180,E1 -8998.168,E2 -8998.168} C_VEL
LIN {X 0,Y 439.768,Z 57.707,A -85,B 0,C 180,E1 -9000,E2 -9000} C_VEL
LIN {X 0,Y 439.644,Z 57.717,A -85,B 0,C 180,E1 -9002.749,E2 -9002.749} C_VEL
LIN {X 0,Y 439.571,Z 57.726,A -85,B 0,C 180,E1 -9006.426,E2 -9006.426} C_VEL
LIN {X 0,Y 439.5,Z 57.738,A -85,B 0,C 180,E1 -9009.202,E2 -9009.202} C_VEL
LIN {X 0,Y 439.471,Z 57.741,A -85,B 0,C 180,E1 -9012.938,E2 -9012.938} C_VEL
LIN {X 0,Y 439.451,Z 57.741,A -85,B 0,C 180,E1 -9016.348,E2 -9016.348} C_VEL
LIN {X 0,Y 439.407,Z 57.749,A -85,B 0,C 180,E1 -9019.626,E2 -9019.626} C_VEL
LIN {X 0,Y 439.369,Z 57.753,A -85,B 0,C 180,E1 -9022.575,E2 -9022.575} C_VEL
LIN {X 0,Y 439.385,Z 57.75,A -85,B 0,C 180,E1 -9025.586,E2 -9025.586} C_VEL
LIN {X 0,Y 439.405,Z 57.752,A -85,B 0,C 180,E1 -9028.675,E2 -9028.675} C_VEL
LIN {X 0,Y 439.373,Z 57.752,A -85,B 0,C 180,E1 -9032.03,E2 -9032.03} C_VEL
LIN {X 0,Y 439.396,Z 57.748,A -85,B 0,C 180,E1 -9035.34,E2 -9035.34} C_VEL
LIN {X 0,Y 439.379,Z 57.756,A -85,B 0,C 180,E1 -9038.596,E2 -9038.596} C_VEL
LIN {X 0,Y 439.392,Z 57.748,A -85,B 0,C 180,E1 -9041.257,E2 -9041.257} C_VEL
LIN {X 0,Y 439.402,Z 57.749,A -85,B 0,C 180,E1 -9044.729,E2 -9044.729} C_VEL
LIN {X 0,Y 439.388,Z 57.752,A -85,B 0,C 180,E1 -9047.794,E2 -9047.794} C_VEL
LIN {X 0,Y 439.392,Z 57.754,A -85,B 0,C 180,E1 -9050.223,E2 -9050.223} C_VEL
LIN {X 0,Y 439.375,Z 57.755,A -85,B 0,C 180,E1 -9053.712,E2 -9053.712} C_VEL
LIN {X 0,Y 439.374,Z 57.751,A -85,B 0,C 180,E1 -9057.054,E2 -9057.054} C_VEL
LIN {X 0,Y 439.385,Z 57.755,A -85,B 0,C 180,E1 -9060.274,E2 -9060.274} C_VEL
LIN {X 0,Y 439.517,Z 57.883,A -85,B 0,C 180,E1 -9062.631,E2 -9062.631} C_VEL
LIN {X 0,Y 441.915,Z 70.563,A -85,B 0,C 180,E1 -9065.027,E2 -9065.027} C_VEL
LIN {X 0,Y 441.31,Z 84.848,A -85,B 0,C 180,E1 -9067.529,E2 -9067.529} C_VEL
LIN {X 0,Y 440.393,Z 105.748,A -85,B 0,C 180,E1 -9071.146,E2 -9071.146} C_VEL
LIN {X 0,Y 440.113,Z 111.558,A -85,B 0,C 180,E1 -9072.127,E2 -9072.127} C_VEL
LIN {X 0,Y 443.394,Z 136.386,A -85,B 0,C 180,E1 -9072.651,E2 -9072.651} C_VEL
LIN {X 0,Y 442.71,Z 219.861,A -85,B 0,C 180,E1 -9074.018,E2 -9074.018} C_VEL
LIN {X 0,Y 442.214,Z 233.333,A -85,B 0,C 180,E1 -9074.414,E2 -9074.414} C_VEL
LIN {X 0,Y 441.672,Z 246.761,A -85,B 0,C 180,E1 -9075.014,E2 -9075.014} C_VEL
LIN {X 0,Y 441.127,Z 258.014,A -85,B 0,C 180,E1 -9075.703,E2 -9075.703} C_VEL
LIN {X 0,Y 440.512,Z 269.623,A -85,B 0,C 180,E1 -9076.617,E2 -9076.617} C_VEL
LIN {X 0,Y 439.908,Z 280.218,A -85,B 0,C 180,E1 -9077.662,E2 -9077.662} C_VEL
LIN {X 0,Y 439.48,Z 288.818,A -85,B 0,C 180,E1 -9078.703,E2 -9078.703} C_VEL
LIN {X 0,Y 438.947,Z 298.12,A -85,B 0,C 180,E1 -9080.089,E2 -9080.089} C_VEL
LIN {X 0,Y 438.671,Z 305.602,A -85,B 0,C 180,E1 -9081.477,E2 -9081.477} C_VEL
LIN {X 0,Y 438.443,Z 312.476,A -85,B 0,C 180,E1 -9083.095,E2 -9083.095} C_VEL
LIN {X 0,Y 438.355,Z 317.002,A -85,B 0,C 180,E1 -9084.48,E2 -9084.48} C_VEL
LIN {X 0,Y 438.347,Z 319.388,A -85,B 0,C 180,E1 -9085.402,E2 -9085.402} C_VEL
LIN {X 0,Y 438.365,Z 321.339,A -85,B 0,C 180,E1 -9086.323,E2 -9086.323} C_VEL
LIN {X 0,Y 438.406,Z 322.862,A -85,B 0,C 180,E1 -9087.243,E2 -9087.243} C_VEL
LIN {X 0,Y 438.38,Z 324.591,A -85,B 0,C 180,E1 -9089.081,E2 -9089.081} C_VEL
LIN {X 0,Y 438.359,Z 324.867,A -85,B 0,C 180,E1 -9090,E2 -9090} C_VEL
LIN {X 0,Y 438.349,Z 324.749,A -85,B 0,C 180,E1 -9090.919,E2 -9090.919} C_VEL
LIN {X 0,Y 438.4,Z 323.249,A -85,B 0,C 180,E1 -9092.757,E2 -9092.757} C_VEL
LIN {X 0,Y 438.332,Z 321.901,A -85,B 0,C 180,E1 -9093.677,E2 -9093.677} C_VEL
LIN {X 0,Y 438.367,Z 319.065,A -85,B 0,C 180,E1 -9095.059,E2 -9095.059} C_VEL
LIN {X 0,Y 438.369,Z 315.203,A -85,B 0,C 180,E1 -9096.444,E2 -9096.444} C_VEL
LIN {X 0,Y 438.588,Z 310.228,A -85,B 0,C 180,E1 -9097.828,E2 -9097.828} C_VEL
LIN {X 0,Y 438.841,Z 303.986,A -85,B 0,C 180,E1 -9099.216,E2 -9099.216} C_VEL
LIN {X 0,Y 439.271,Z 296.228,A -85,B 0,C 180,E1 -9100.602,E2 -9100.602} C_VEL
LIN {X 0,Y 439.977,Z 286.531,A -85,B 0,C 180,E1 -9101.985,E2 -9101.985} C_VEL
LIN {X 0,Y 440.571,Z 276.323,A -85,B 0,C 180,E1 -9103.163,E2 -9103.163} C_VEL
LIN {X 0,Y 441.336,Z 265.302,A -85,B 0,C 180,E1 -9104.172,E2 -9104.172} C_VEL
LIN {X 0,Y 442.037,Z 254.311,A -85,B 0,C 180,E1 -9104.973,E2 -9104.973} C_VEL
LIN {X 0,Y 442.726,Z 242.16,A -85,B 0,C 180,E1 -9105.656,E2 -9105.656} C_VEL
LIN {X 0,Y 443.352,Z 230.404,A -85,B 0,C 180,E1 -9106.135,E2 -9106.135} C_VEL
LIN {X 0,Y 443.736,Z 217.751,A -85,B 0,C 180,E1 -9106.475,E2 -9106.475} C_VEL
LIN {X 0,Y 444.41,Z 135.802,A -85,B 0,C 180,E1 -9107.837,E2 -9107.837} C_VEL
LIN {X 0,Y 441.452,Z 116.353,A -85,B 0,C 180,E1 -9108.307,E2 -9108.307} C_VEL
LIN {X 0,Y 440.577,Z 111.017,A -85,B 0,C 180,E1 -9108.449,E2 -9108.449} C_VEL
LIN {X 0,Y 441.549,Z 92.512,A -85,B 0,C 180,E1 -9111.72,E2 -9111.72} C_VEL
LIN {X 0,Y 442.692,Z 74.124,A -85,B 0,C 180,E1 -9115.018,E2 -9115.018} C_VEL
LIN {X 0,Y 441.456,Z 66.72,A -85,B 0,C 180,E1 -9116.472,E2 -9116.472} C_VEL
LIN {X 0,Y 439.446,Z 57.748,A -85,B 0,C 180,E1 -9118.311,E2 -9118.311} C_VEL
LIN {X 0,Y 439.375,Z 57.755,A -85,B 0,C 180,E1 -9121.861,E2 -9121.861} C_VEL
LIN {X 0,Y 439.399,Z 57.75,A -85,B 0,C 180,E1 -9125.156,E2 -9125.156} C_VEL
LIN {X 0,Y 439.381,Z 57.748,A -85,B 0,C 180,E1 -9128.595,E2 -9128.595} C_VEL
LIN {X 0,Y 439.391,Z 57.751,A -85,B 0,C 180,E1 -9131.257,E2 -9131.257} C_VEL
LIN {X 0,Y 439.403,Z 57.744,A -85,B 0,C 180,E1 -9134.729,E2 -9134.729} C_VEL
LIN {X 0,Y 439.399,Z 57.75,A -85,B 0,C 180,E1 -9137.796,E2 -9137.796} C_VEL
LIN {X 0,Y 439.398,Z 57.744,A -85,B 0,C 180,E1 -9140.224,E2 -9140.224} C_VEL
LIN {X 0,Y 439.376,Z 57.752,A -85,B 0,C 180,E1 -9143.713,E2 -9143.713} C_VEL
LIN {X 0,Y 439.375,Z 57.752,A -85,B 0,C 180,E1 -9147.054,E2 -9147.054} C_VEL
LIN {X 0,Y 439.386,Z 57.747,A -85,B 0,C 180,E1 -9150.274,E2 -9150.274} C_VEL
LIN {X 0,Y 439.432,Z 57.742,A -85,B 0,C 180,E1 -9153.396,E2 -9153.396} C_VEL
LIN {X 0,Y 439.39,Z 57.753,A -85,B 0,C 180,E1 -9156.43,E2 -9156.43} C_VEL
LIN {X 0,Y 439.392,Z 57.749,A -85,B 0,C 180,E1 -9159.397,E2 -9159.397} C_VEL
LIN {X 0,Y 439.434,Z 57.746,A -85,B 0,C 180,E1 -9162.31,E2 -9162.31} C_VEL
LIN {X 0,Y 439.452,Z 57.742,A -85,B 0,C 180,E1 -9165.174,E2 -9165.174} C_VEL
LIN {X 0,Y 439.488,Z 57.736,A -85,B 0,C 180,E1 -9168.001,E2 -9168.001} C_VEL
LIN {X 0,Y 439.552,Z 57.731,A -85,B 0,C 180,E1 -9171.726,E2 -9171.726} C_VEL
LIN {X 0,Y 439.622,Z 57.722,A -85,B 0,C 180,E1 -9174.496,E2 -9174.496} C_VEL
LIN {X 0,Y 439.637,Z 57.716,A -85,B 0,C 180,E1 -9178.168,E2 -9178.168} C_VEL
LIN {X 0,Y 439.767,Z 57.708,A -85,B 0,C 180,E1 -9180,E2 -9180} C_VEL
LIN {X 0,Y 439.643,Z 57.715,A -85,B 0,C 180,E1 -9182.749,E2 -9182.749} C_VEL
LIN {X 0,Y 439.604,Z 57.723,A -85,B 0,C 180,E1 -9186.425,E2 -9186.425} C_VEL
LIN {X 0,Y 439.499,Z 57.734,A -85,B 0,C 180,E1 -9189.202,E2 -9189.202} C_VEL
LIN {X 0,Y 439.469,Z 57.742,A -85,B 0,C 180,E1 -9192.937,E2 -9192.937} C_VEL
LIN {X 0,Y 439.45,Z 57.743,A -85,B 0,C 180,E1 -9196.348,E2 -9196.348} C_VEL
LIN {X 0,Y 439.405,Z 57.748,A -85,B 0,C 180,E1 -9199.626,E2 -9199.626} C_VEL
LIN {X 0,Y 439.368,Z 57.755,A -85,B 0,C 180,E1 -9202.575,E2 -9202.575} C_VEL
LIN {X 0,Y 439.385,Z 57.75,A -85,B 0,C 180,E1 -9205.586,E2 -9205.586} C_VEL
LIN {X 0,Y 439.403,Z 57.754,A -85,B 0,C 180,E1 -9208.674,E2 -9208.674} C_VEL
LIN {X 0,Y 439.371,Z 57.753,A -85,B 0,C 180,E1 -9212.03,E2 -9212.03} C_VEL
LIN {X 0,Y 439.393,Z 57.75,A -85,B 0,C 180,E1 -9215.339,E2 -9215.339} C_VEL
LIN {X 0,Y 439.365,Z 57.756,A -85,B 0,C 180,E1 -9218.597,E2 -9218.597} C_VEL
LIN {X 0,Y 439.382,Z 57.743,A -85,B 0,C 180,E1 -9221.255,E2 -9221.255} C_VEL
LIN {X 0,Y 439.4,Z 57.751,A -85,B 0,C 180,E1 -9224.729,E2 -9224.729} C_VEL
LIN {X 0,Y 439.385,Z 57.756,A -85,B 0,C 180,E1 -9227.794,E2 -9227.794} C_VEL
LIN {X 0,Y 439.359,Z 57.757,A -85,B 0,C 180,E1 -9230.22,E2 -9230.22} C_VEL
LIN {X 0,Y 439.372,Z 57.759,A -85,B 0,C 180,E1 -9233.712,E2 -9233.712} C_VEL
LIN {X 0,Y 439.373,Z 57.76,A -85,B 0,C 180,E1 -9237.054,E2 -9237.054} C_VEL
LIN {X 0,Y 439.426,Z 57.892,A -85,B 0,C 180,E1 -9239.216,E2 -9239.216} C_VEL
LIN {X 0,Y 441.106,Z 66.852,A -85,B 0,C 180,E1 -9241.446,E2 -9241.446} C_VEL
LIN {X 0,Y 441.185,Z 67.845,A -85,B 0,C 180,E1 -9241.643,E2 -9241.643} C_VEL
LIN {X 0,Y 445.056,Z 83.512,A -85,B 0,C 180,E1 -9242.103,E2 -9242.103} C_VEL
LIN {X 0,Y 443.97,Z 174.928,A -85,B 0,C 180,E1 -9243.626,E2 -9243.626} C_VEL
LIN {X 0,Y 443.703,Z 188.367,A -85,B 0,C 180,E1 -9244.052,E2 -9244.052} C_VEL
LIN {X 0,Y 443.302,Z 201.19,A -85,B 0,C 180,E1 -9244.656,E2 -9244.656} C_VEL
LIN {X 0,Y 442.711,Z 212.559,A -85,B 0,C 180,E1 -9245.377,E2 -9245.377} C_VEL
LIN {X 0,Y 441.997,Z 224.23,A -85,B 0,C 180,E1 -9246.329,E2 -9246.329} C_VEL
LIN {X 0,Y 441.392,Z 233.866,A -85,B 0,C 180,E1 -9247.312,E2 -9247.312} C_VEL
LIN {X 0,Y 440.765,Z 243.203,A -85,B 0,C 180,E1 -9248.486,E2 -9248.486} C_VEL
LIN {X 0,Y 440.194,Z 250.982,A -85,B 0,C 180,E1 -9249.68,E2 -9249.68} C_VEL
LIN {X 0,Y 439.697,Z 257.246,A -85,B 0,C 180,E1 -9250.84,E2 -9250.84} C_VEL
LIN {X 0,Y 438.798,Z 260.385,A -85,B 0,C 180,E1 -9251.487,E2 -9251.487} C_VEL
LIN {X 0,Y 435.646,Z 265.115,A -85,B 0,C 180,E1 -9252.555,E2 -9252.555} C_VEL
LIN {X 0,Y 432.551,Z 269.134,A -85,B 0,C 180,E1 -9253.68,E2 -9253.68} C_VEL
LIN {X 0,Y 431.75,Z 271.173,A -85,B 0,C 180,E1 -9254.405,E2 -9254.405} C_VEL
LIN {X 0,Y 431.509,Z 274.308,A -85,B 0,C 180,E1 -9255.859,E2 -9255.859} C_VEL
LIN {X 0,Y 431.41,Z 275.826,A -85,B 0,C 180,E1 -9256.816,E2 -9256.816} C_VEL
LIN {X 0,Y 431.338,Z 276.943,A -85,B 0,C 180,E1 -9257.852,E2 -9257.852} C_VEL
LIN {X 0,Y 431.26,Z 277.788,A -85,B 0,C 180,E1 -9259.673,E2 -9259.673} C_VEL
LIN {X 0,Y 431.254,Z 277.642,A -85,B 0,C 180,E1 -9260.621,E2 -9260.621} C_VEL
LIN {X 0,Y 431.349,Z 276.099,A -85,B 0,C 180,E1 -9262.511,E2 -9262.511} C_VEL
LIN {X 0,Y 431.468,Z 274.641,A -85,B 0,C 180,E1 -9263.516,E2 -9263.516} C_VEL
LIN {X 0,Y 431.514,Z 271.89,A -85,B 0,C 180,E1 -9264.861,E2 -9264.861} C_VEL
LIN {X 0,Y 431.747,Z 268.011,A -85,B 0,C 180,E1 -9266.267,E2 -9266.267} C_VEL
LIN {X 0,Y 431.946,Z 263.025,A -85,B 0,C 180,E1 -9267.669,E2 -9267.669} C_VEL
LIN {X 0,Y 432.304,Z 256.758,A -85,B 0,C 180,E1 -9269.069,E2 -9269.069} C_VEL
LIN {X 0,Y 432.777,Z 248.921,A -85,B 0,C 180,E1 -9270.465,E2 -9270.465} C_VEL
LIN {X 0,Y 433.186,Z 240.962,A -85,B 0,C 180,E1 -9271.627,E2 -9271.627} C_VEL
LIN {X 0,Y 433.872,Z 231.227,A -85,B 0,C 180,E1 -9272.785,E2 -9272.785} C_VEL
LIN {X 0,Y 434.433,Z 221.691,A -85,B 0,C 180,E1 -9273.71,E2 -9273.71} C_VEL
LIN {X 0,Y 435.007,Z 211.433,A -85,B 0,C 180,E1 -9274.517,E2 -9274.517} C_VEL
LIN {X 0,Y 435.457,Z 199.211,A -85,B 0,C 180,E1 -9275.267,E2 -9275.267} C_VEL
LIN {X 0,Y 435.774,Z 186.392,A -85,B 0,C 180,E1 -9275.843,E2 -9275.843} C_VEL
LIN {X 0,Y 436.061,Z 173.888,A -85,B 0,C 180,E1 -9276.217,E2 -9276.217} C_VEL
LIN {X 0,Y 436.962,Z 83.982,A -85,B 0,C 180,E1 -9277.71,E2 -9277.71} C_VEL
LIN {X 0,Y 433.738,Z 67.583,A -85,B 0,C 180,E1 -9278.116,E2 -9278.116} C_VEL
LIN {X 0,Y 432.776,Z 60.393,A -85,B 0,C 180,E1 -9279.818,E2 -9279.818} C_VEL
LIN {X 0,Y 432.408,Z 58.626,A -85,B 0,C 180,E1 -9280.299,E2 -9280.299} C_VEL
LIN {X 0,Y 432.402,Z 58.623,A -85,B 0,C 180,E1 -9283.153,E2 -9283.153} C_VEL
LIN {X 0,Y 432.414,Z 58.625,A -85,B 0,C 180,E1 -9286.479,E2 -9286.479} C_VEL
LIN {X 0,Y 432.341,Z 58.629,A -85,B 0,C 180,E1 -9289.961,E2 -9289.961} C_VEL
LIN {X 0,Y 432.319,Z 58.63,A -85,B 0,C 180,E1 -9292.964,E2 -9292.964} C_VEL
LIN {X 0,Y 432.363,Z 58.63,A -85,B 0,C 180,E1 -9296.033,E2 -9296.033} C_VEL
LIN {X 0,Y 432.345,Z 58.626,A -85,B 0,C 180,E1 -9299.188,E2 -9299.188} C_VEL
LIN {X 0,Y 432.325,Z 58.63,A -85,B 0,C 180,E1 -9302.443,E2 -9302.443} C_VEL
LIN {X 0,Y 432.348,Z 58.631,A -85,B 0,C 180,E1 -9305.632,E2 -9305.632} C_VEL
LIN {X 0,Y 432.355,Z 58.625,A -85,B 0,C 180,E1 -9308.717,E2 -9308.717} C_VEL
LIN {X 0,Y 432.336,Z 58.632,A -85,B 0,C 180,E1 -9311.797,E2 -9311.797} C_VEL
LIN {X 0,Y 432.336,Z 58.628,A -85,B 0,C 180,E1 -9314.348,E2 -9314.348} C_VEL
LIN {X 0,Y 432.322,Z 58.632,A -85,B 0,C 180,E1 -9317.016,E2 -9317.016} C_VEL
LIN {X 0,Y 432.336,Z 58.629,A -85,B 0,C 180,E1 -9319.821,E2 -9319.821} C_VEL
LIN {X 0,Y 432.31,Z 58.636,A -85,B 0,C 180,E1 -9323.022,E2 -9323.022} C_VEL
LIN {X 0,Y 432.363,Z 58.624,A -85,B 0,C 180,E1 -9325.997,E2 -9325.997} C_VEL
LIN {X 0,Y 432.351,Z 58.627,A -85,B 0,C 180,E1 -9329.49,E2 -9329.49} C_VEL
LIN {X 0,Y 432.395,Z 58.626,A -85,B 0,C 180,E1 -9332.929,E2 -9332.929} C_VEL
LIN {X 0,Y 432.375,Z 58.623,A -85,B 0,C 180,E1 -9336.024,E2 -9336.024} C_VEL
LIN {X 0,Y 432.354,Z 58.627,A -85,B 0,C 180,E1 -9339.046,E2 -9339.046} C_VEL
LIN {X 0,Y 432.377,Z 58.624,A -85,B 0,C 180,E1 -9342.011,E2 -9342.011} C_VEL
LIN {X 0,Y 432.4,Z 58.621,A -85,B 0,C 180,E1 -9344.927,E2 -9344.927} C_VEL
LIN {X 0,Y 432.464,Z 58.613,A -85,B 0,C 180,E1 -9347.804,E2 -9347.804} C_VEL
LIN {X 0,Y 432.486,Z 58.61,A -85,B 0,C 180,E1 -9351.59,E2 -9351.59} C_VEL
LIN {X 0,Y 432.599,Z 58.598,A -85,B 0,C 180,E1 -9354.406,E2 -9354.406} C_VEL
LIN {X 0,Y 432.607,Z 58.598,A -85,B 0,C 180,E1 -9358.138,E2 -9358.138} C_VEL
LIN {X 0,Y 432.737,Z 58.583,A -85,B 0,C 180,E1 -9360,E2 -9360} C_VEL
LIN {X 0,Y 432.596,Z 58.595,A -85,B 0,C 180,E1 -9362.794,E2 -9362.794} C_VEL
LIN {X 0,Y 432.585,Z 58.603,A -85,B 0,C 180,E1 -9365.594,E2 -9365.594} C_VEL
LIN {X 0,Y 432.469,Z 58.611,A -85,B 0,C 180,E1 -9368.41,E2 -9368.41} C_VEL
LIN {X 0,Y 432.464,Z 58.612,A -85,B 0,C 180,E1 -9372.197,E2 -9372.197} C_VEL
LIN {X 0,Y 432.435,Z 58.615,A -85,B 0,C 180,E1 -9376.039,E2 -9376.039} C_VEL
LIN {X 0,Y 432.391,Z 58.624,A -85,B 0,C 180,E1 -9379.485,E2 -9379.485} C_VEL
LIN {X 0,Y 432.322,Z 58.636,A -85,B 0,C 180,E1 -9382.964,E2 -9382.964} C_VEL
LIN {X 0,Y 432.344,Z 58.633,A -85,B 0,C 180,E1 -9385.002,E2 -9385.002} C_VEL
LIN {X 0,Y 432.352,Z 58.626,A -85,B 0,C 180,E1 -9388.126,E2 -9388.126} C_VEL
LIN {X 0,Y 432.325,Z 58.63,A -85,B 0,C 180,E1 -9391.346,E2 -9391.346} C_VEL
LIN {X 0,Y 432.341,Z 58.633,A -85,B 0,C 180,E1 -9394.677,E2 -9394.677} C_VEL
LIN {X 0,Y 432.339,Z 58.63,A -85,B 0,C 180,E1 -9398.15,E2 -9398.15} C_VEL
LIN {X 0,Y 432.336,Z 58.628,A -85,B 0,C 180,E1 -9401.602,E2 -9401.602} C_VEL
LIN {X 0,Y 432.337,Z 58.633,A -85,B 0,C 180,E1 -9404.347,E2 -9404.347} C_VEL
LIN {X 0,Y 432.32,Z 58.63,A -85,B 0,C 180,E1 -9407.016,E2 -9407.016} C_VEL
LIN {X 0,Y 432.316,Z 58.634,A -85,B 0,C 180,E1 -9409.824,E2 -9409.824} C_VEL
LIN {X 0,Y 432.307,Z 58.631,A -85,B 0,C 180,E1 -9413.022,E2 -9413.022} C_VEL
LIN {X 0,Y 432.36,Z 58.63,A -85,B 0,C 180,E1 -9415.997,E2 -9415.997} C_VEL
LIN {X 0,Y 432.35,Z 58.63,A -85,B 0,C 180,E1 -9419.49,E2 -9419.49} C_VEL
LIN {X 0,Y 432.458,Z 58.635,A -85,B 0,C 180,E1 -9422.408,E2 -9422.408} C_VEL
LIN {X 0,Y 434.876,Z 71.194,A -85,B 0,C 180,E1 -9424.825,E2 -9424.825} C_VEL
LIN {X 0,Y 434.791,Z 77.226,A -85,B 0,C 180,E1 -9425.911,E2 -9425.911} C_VEL
LIN {X 0,Y 433.755,Z 96.782,A -85,B 0,C 180,E1 -9429.365,E2 -9429.365} C_VEL
LIN {X 0,Y 433.115,Z 111.022,A -85,B 0,C 180,E1 -9431.859,E2 -9431.859} C_VEL
LIN {X 0,Y 436.558,Z 138.563,A -85,B 0,C 180,E1 -9432.453,E2 -9432.453} C_VEL
LIN {X 0,Y 435.786,Z 220.294,A -85,B 0,C 180,E1 -9433.817,E2 -9433.817} C_VEL
LIN {X 0,Y 435.278,Z 233.482,A -85,B 0,C 180,E1 -9434.219,E2 -9434.219} C_VEL
LIN {X 0,Y 434.794,Z 245.647,A -85,B 0,C 180,E1 -9434.772,E2 -9434.772} C_VEL
LIN {X 0,Y 434.182,Z 257.107,A -85,B 0,C 180,E1 -9435.469,E2 -9435.469} C_VEL
LIN {X 0,Y 433.583,Z 267.985,A -85,B 0,C 180,E1 -9436.323,E2 -9436.323} C_VEL
LIN {X 0,Y 432.949,Z 279.496,A -85,B 0,C 180,E1 -9437.46,E2 -9437.46} C_VEL
LIN {X 0,Y 432.476,Z 288.154,A -85,B 0,C 180,E1 -9438.517,E2 -9438.517} C_VEL
LIN {X 0,Y 431.969,Z 296.125,A -85,B 0,C 180,E1 -9439.69,E2 -9439.69} C_VEL
LIN {X 0,Y 431.608,Z 303.91,A -85,B 0,C 180,E1 -9441.101,E2 -9441.101} C_VEL
LIN {X 0,Y 431.414,Z 310.158,A -85,B 0,C 180,E1 -9442.511,E2 -9442.511} C_VEL
LIN {X 0,Y 431.25,Z 314.674,A -85,B 0,C 180,E1 -9443.778,E2 -9443.778} C_VEL
LIN {X 0,Y 431.277,Z 318.925,A -85,B 0,C 180,E1 -9445.326,E2 -9445.326} C_VEL
LIN {X 0,Y 431.267,Z 320.887,A -85,B 0,C 180,E1 -9446.262,E2 -9446.262} C_VEL
LIN {X 0,Y 431.333,Z 322.431,A -85,B 0,C 180,E1 -9447.198,E2 -9447.198} C_VEL
LIN {X 0,Y 431.29,Z 323.51,A -85,B 0,C 180,E1 -9448.132,E2 -9448.132} C_VEL
LIN {X 0,Y 431.289,Z 324.189,A -85,B 0,C 180,E1 -9449.066,E2 -9449.066} C_VEL
LIN {X 0,Y 431.297,Z 324.478,A -85,B 0,C 180,E1 -9450,E2 -9450} C_VEL
LIN {X 0,Y 431.26,Z 324.374,A -85,B 0,C 180,E1 -9450.934,E2 -9450.934} C_VEL
LIN {X 0,Y 431.269,Z 323.841,A -85,B 0,C 180,E1 -9451.868,E2 -9451.868} C_VEL
LIN {X 0,Y 431.326,Z 322.906,A -85,B 0,C 180,E1 -9452.802,E2 -9452.802} C_VEL
LIN {X 0,Y 431.27,Z 319.828,A -85,B 0,C 180,E1 -9454.674,E2 -9454.674} C_VEL
LIN {X 0,Y 431.25,Z 315.931,A -85,B 0,C 180,E1 -9456.222,E2 -9456.222} C_VEL
LIN {X 0,Y 431.437,Z 311.782,A -85,B 0,C 180,E1 -9457.488,E2 -9457.488} C_VEL
LIN {X 0,Y 431.725,Z 304.894,A -85,B 0,C 180,E1 -9459.133,E2 -9459.133} C_VEL
LIN {X 0,Y 432.159,Z 297.447,A -85,B 0,C 180,E1 -9460.542,E2 -9460.542} C_VEL
LIN {X 0,Y 432.885,Z 288.215,A -85,B 0,C 180,E1 -9461.947,E2 -9461.947} C_VEL
LIN {X 0,Y 433.497,Z 278.647,A -85,B 0,C 180,E1 -9463.119,E2 -9463.119} C_VEL
LIN {X 0,Y 434.256,Z 268.067,A -85,B 0,C 180,E1 -9464.169,E2 -9464.169} C_VEL
LIN {X 0,Y 435.069,Z 256.266,A -85,B 0,C 180,E1 -9465.099,E2 -9465.099} C_VEL
LIN {X 0,Y 435.884,Z 243.644,A -85,B 0,C 180,E1 -9465.848,E2 -9465.848} C_VEL
LIN {X 0,Y 436.49,Z 232.584,A -85,B 0,C 180,E1 -9466.336,E2 -9466.336} C_VEL
LIN {X 0,Y 436.963,Z 219.281,A -85,B 0,C 180,E1 -9466.738,E2 -9466.738} C_VEL
LIN {X 0,Y 437.824,Z 137.281,A -85,B 0,C 180,E1 -9468.123,E2 -9468.123} C_VEL
LIN {X 0,Y 434.886,Z 117.66,A -85,B 0,C 180,E1 -9468.607,E2 -9468.607} C_VEL
LIN {X 0,Y 433.664,Z 110.661,A -85,B 0,C 180,E1 -9468.792,E2 -9468.792} C_VEL
LIN {X 0,Y 434.72,Z 92.378,A -85,B 0,C 180,E1 -9472.079,E2 -9472.079} C_VEL
LIN {X 0,Y 435.79,Z 75.089,A -85,B 0,C 180,E1 -9475.241,E2 -9475.241} C_VEL
LIN {X 0,Y 433.939,Z 65.268,A -85,B 0,C 180,E1 -9477.228,E2 -9477.228} C_VEL
LIN {X 0,Y 432.379,Z 58.625,A -85,B 0,C 180,E1 -9478.63,E2 -9478.63} C_VEL
LIN {X 0,Y 432.323,Z 58.63,A -85,B 0,C 180,E1 -9481.346,E2 -9481.346} C_VEL
LIN {X 0,Y 432.34,Z 58.63,A -85,B 0,C 180,E1 -9484.677,E2 -9484.677} C_VEL
LIN {X 0,Y 432.34,Z 58.629,A -85,B 0,C 180,E1 -9488.15,E2 -9488.15} C_VEL
LIN {X 0,Y 432.336,Z 58.633,A -85,B 0,C 180,E1 -9491.602,E2 -9491.602} C_VEL
LIN {X 0,Y 432.336,Z 58.626,A -85,B 0,C 180,E1 -9494.347,E2 -9494.347} C_VEL
LIN {X 0,Y 432.323,Z 58.629,A -85,B 0,C 180,E1 -9497.016,E2 -9497.016} C_VEL
LIN {X 0,Y 432.336,Z 58.626,A -85,B 0,C 180,E1 -9499.821,E2 -9499.821} C_VEL
LIN {X 0,Y 432.309,Z 58.632,A -85,B 0,C 180,E1 -9503.022,E2 -9503.022} C_VEL
LIN {X 0,Y 432.361,Z 58.622,A -85,B 0,C 180,E1 -9505.997,E2 -9505.997} C_VEL
LIN {X 0,Y 432.351,Z 58.625,A -85,B 0,C 180,E1 -9509.49,E2 -9509.49} C_VEL
LIN {X 0,Y 432.394,Z 58.625,A -85,B 0,C 180,E1 -9512.928,E2 -9512.928} C_VEL
LIN {X 0,Y 432.374,Z 58.624,A -85,B 0,C 180,E1 -9516.023,E2 -9516.023} C_VEL
LIN {X 0,Y 432.354,Z 58.628,A -85,B 0,C 180,E1 -9519.046,E2 -9519.046} C_VEL
LIN {X 0,Y 432.381,Z 58.623,A -85,B 0,C 180,E1 -9522.011,E2 -9522.011} C_VEL
LIN {X 0,Y 432.4,Z 58.622,A -85,B 0,C 180,E1 -9524.926,E2 -9524.926} C_VEL
LIN {X 0,Y 432.463,Z 58.61,A -85,B 0,C 180,E1 -9527.803,E2 -9527.803} C_VEL
LIN {X 0,Y 432.496,Z 58.609,A -85,B 0,C 180,E1 -9531.59,E2 -9531.59} C_VEL
LIN {X 0,Y 432.599,Z 58.598,A -85,B 0,C 180,E1 -9534.406,E2 -9534.406} C_VEL
LIN {X 0,Y 432.606,Z 58.592,A -85,B 0,C 180,E1 -9538.138,E2 -9538.138} C_VEL
LIN {X 0,Y 432.736,Z 58.584,A -85,B 0,C 180,E1 -9540,E2 -9540} C_VEL
LIN {X 0,Y 432.594,Z 58.593,A -85,B 0,C 180,E1 -9542.794,E2 -9542.794} C_VEL
LIN {X 0,Y 432.554,Z 58.601,A -85,B 0,C 180,E1 -9546.53,E2 -9546.53} C_VEL
LIN {X 0,Y 432.443,Z 58.613,A -85,B 0,C 180,E1 -9549.353,E2 -9549.353} C_VEL
LIN {X 0,Y 432.435,Z 58.617,A -85,B 0,C 180,E1 -9552.803,E2 -9552.803} C_VEL
LIN {X 0,Y 432.415,Z 58.619,A -85,B 0,C 180,E1 -9556.478,E2 -9556.478} C_VEL
LIN {X 0,Y 432.341,Z 58.627,A -85,B 0,C 180,E1 -9559.96,E2 -9559.96} C_VEL
LIN {X 0,Y 432.322,Z 58.631,A -85,B 0,C 180,E1 -9562.964,E2 -9562.964} C_VEL
LIN {X 0,Y 432.344,Z 58.632,A -85,B 0,C 180,E1 -9565.002,E2 -9565.002} C_VEL
LIN {X 0,Y 432.35,Z 58.626,A -85,B 0,C 180,E1 -9568.125,E2 -9568.125} C_VEL
LIN {X 0,Y 432.323,Z 58.63,A -85,B 0,C 180,E1 -9571.346,E2 -9571.346} C_VEL
LIN {X 0,Y 432.339,Z 58.633,A -85,B 0,C 180,E1 -9574.677,E2 -9574.677} C_VEL
LIN {X 0,Y 432.332,Z 58.634,A -85,B 0,C 180,E1 -9578.15,E2 -9578.15} C_VEL
LIN {X 0,Y 432.326,Z 58.624,A -85,B 0,C 180,E1 -9581.6,E2 -9581.6} C_VEL
LIN {X 0,Y 432.335,Z 58.633,A -85,B 0,C 180,E1 -9584.347,E2 -9584.347} C_VEL
LIN {X 0,Y 432.317,Z 58.633,A -85,B 0,C 180,E1 -9587.016,E2 -9587.016} C_VEL
LIN {X 0,Y 432.315,Z 58.636,A -85,B 0,C 180,E1 -9589.824,E2 -9589.824} C_VEL
LIN {X 0,Y 432.305,Z 58.636,A -85,B 0,C 180,E1 -9593.022,E2 -9593.022} C_VEL
LIN {X 0,Y 432.358,Z 58.63,A -85,B 0,C 180,E1 -9595.997,E2 -9595.997} C_VEL
LIN {X 0,Y 432.356,Z 58.708,A -85,B 0,C 180,E1 -9598.924,E2 -9598.924} C_VEL
LIN {X 0,Y 434.188,Z 68.085,A -85,B 0,C 180,E1 -9601.286,E2 -9601.286} C_VEL
LIN {X 0,Y 438.303,Z 83.927,A -85,B 0,C 180,E1 -9601.774,E2 -9601.774} C_VEL
LIN {X 0,Y 438.384,Z 89.839,A -85,B 0,C 180,E1 -9601.88,E2 -9601.88} C_VEL
LIN {X 0,Y 437.276,Z 175.043,A -85,B 0,C 180,E1 -9603.319,E2 -9603.319} C_VEL
LIN {X 0,Y 436.994,Z 188.559,A -85,B 0,C 180,E1 -9603.751,E2 -9603.751} C_VEL
LIN {X 0,Y 436.595,Z 201.164,A -85,B 0,C 180,E1 -9604.349,E2 -9604.349} C_VEL
LIN {X 0,Y 435.935,Z 213.032,A -85,B 0,C 180,E1 -9605.11,E2 -9605.11} C_VEL
LIN {X 0,Y 435.193,Z 224.534,A -85,B 0,C 180,E1 -9606.062,E2 -9606.062} C_VEL
LIN {X 0,Y 434.499,Z 235.028,A -85,B 0,C 180,E1 -9607.157,E2 -9607.157} C_VEL
LIN {X 0,Y 433.798,Z 244.364,A -85,B 0,C 180,E1 -9608.372,E2 -9608.372} C_VEL
LIN {X 0,Y 433.116,Z 253.394,A -85,B 0,C 180,E1 -9609.829,E2 -9609.829} C_VEL
LIN {X 0,Y 432.533,Z 260.538,A -85,B 0,C 180,E1 -9611.282,E2 -9611.282} C_VEL
LIN {X 0,Y 432.033,Z 267.007,A -85,B 0,C 180,E1 -9612.974,E2 -9612.974} C_VEL
LIN {X 0,Y 431.75,Z 271.173,A -85,B 0,C 180,E1 -9614.405,E2 -9614.405} C_VEL
LIN {X 0,Y 430.954,Z 272.988,A -85,B 0,C 180,E1 -9615.144,E2 -9615.144} C_VEL
LIN {X 0,Y 427.912,Z 275.409,A -85,B 0,C 180,E1 -9616.36,E2 -9616.36} C_VEL
LIN {X 0,Y 425.393,Z 276.874,A -85,B 0,C 180,E1 -9617.358,E2 -9617.358} C_VEL
LIN {X 0,Y 424.308,Z 277.621,A -85,B 0,C 180,E1 -9618.138,E2 -9618.138} C_VEL
LIN {X 0,Y 424.216,Z 277.76,A -85,B 0,C 180,E1 -9618.403,E2 -9618.403} C_VEL
LIN {X 0,Y 424.169,Z 278.153,A -85,B 0,C 180,E1 -9619.499,E2 -9619.499} C_VEL
LIN {X 0,Y 424.159,Z 278.07,A -85,B 0,C 180,E1 -9620.463,E2 -9620.463} C_VEL
LIN {X 0,Y 424.181,Z 277.559,A -85,B 0,C 180,E1 -9621.424,E2 -9621.424} C_VEL
LIN {X 0,Y 424.261,Z 276.635,A -85,B 0,C 180,E1 -9622.385,E2 -9622.385} C_VEL
LIN {X 0,Y 424.401,Z 275.066,A -85,B 0,C 180,E1 -9623.508,E2 -9623.508} C_VEL
LIN {X 0,Y 424.442,Z 272.555,A -85,B 0,C 180,E1 -9624.775,E2 -9624.775} C_VEL
LIN {X 0,Y 424.668,Z 268.771,A -85,B 0,C 180,E1 -9626.204,E2 -9626.204} C_VEL
LIN {X 0,Y 424.852,Z 263.888,A -85,B 0,C 180,E1 -9627.63,E2 -9627.63} C_VEL
LIN {X 0,Y 425.221,Z 257.741,A -85,B 0,C 180,E1 -9629.053,E2 -9629.053} C_VEL
LIN {X 0,Y 425.717,Z 250.082,A -85,B 0,C 180,E1 -9630.473,E2 -9630.473} C_VEL
LIN {X 0,Y 426.271,Z 240.508,A -85,B 0,C 180,E1 -9631.89,E2 -9631.89} C_VEL
LIN {X 0,Y 426.914,Z 231.664,A -85,B 0,C 180,E1 -9632.949,E2 -9632.949} C_VEL
LIN {X 0,Y 427.492,Z 222.141,A -85,B 0,C 180,E1 -9633.889,E2 -9633.889} C_VEL
LIN {X 0,Y 428.079,Z 211.901,A -85,B 0,C 180,E1 -9634.709,E2 -9634.709} C_VEL
LIN {X 0,Y 428.553,Z 199.712,A -85,B 0,C 180,E1 -9635.47,E2 -9635.47} C_VEL
LIN {X 0,Y 428.902,Z 186.181,A -85,B 0,C 180,E1 -9636.085,E2 -9636.085} C_VEL
LIN {X 0,Y 429.208,Z 173.171,A -85,B 0,C 180,E1 -9636.464,E2 -9636.464} C_VEL
LIN {X 0,Y 430.106,Z 84.908,A -85,B 0,C 180,E1 -9637.948,E2 -9637.948} C_VEL
LIN {X 0,Y 426.746,Z 67.937,A -85,B 0,C 180,E1 -9638.376,E2 -9638.376} C_VEL
LIN {X 0,Y 425.366,Z 59.503,A -85,B 0,C 180,E1 -9640.472,E2 -9640.472} C_VEL
LIN {X 0,Y 425.367,Z 59.498,A -85,B 0,C 180,E1 -9643.374,E2 -9643.374} C_VEL
LIN {X 0,Y 425.363,Z 59.502,A -85,B 0,C 180,E1 -9646.605,E2 -9646.605} C_VEL
LIN {X 0,Y 425.33,Z 59.501,A -85,B 0,C 180,E1 -9649.636,E2 -9649.636} C_VEL
LIN {X 0,Y 425.289,Z 59.512,A -85,B 0,C 180,E1 -9652.339,E2 -9652.339} C_VEL
LIN {X 0,Y 425.292,Z 59.505,A -85,B 0,C 180,E1 -9655.446,E2 -9655.446} C_VEL
LIN {X 0,Y 425.351,Z 59.499,A -85,B 0,C 180,E1 -9657.558,E2 -9657.558} C_VEL
LIN {X 0,Y 425.29,Z 59.505,A -85,B 0,C 180,E1 -9660.816,E2 -9660.816} C_VEL
LIN {X 0,Y 425.314,Z 59.505,A -85,B 0,C 180,E1 -9664.288,E2 -9664.288} C_VEL
LIN {X 0,Y 425.288,Z 59.512,A -85,B 0,C 180,E1 -9667.694,E2 -9667.694} C_VEL
LIN {X 0,Y 425.286,Z 59.506,A -85,B 0,C 180,E1 -9670.521,E2 -9670.521} C_VEL
LIN {X 0,Y 425.26,Z 59.514,A -85,B 0,C 180,E1 -9673.351,E2 -9673.351} C_VEL
LIN {X 0,Y 425.26,Z 59.509,A -85,B 0,C 180,E1 -9676.649,E2 -9676.649} C_VEL
LIN {X 0,Y 425.289,Z 59.507,A -85,B 0,C 180,E1 -9679.873,E2 -9679.873} C_VEL
LIN {X 0,Y 425.281,Z 59.507,A -85,B 0,C 180,E1 -9682.489,E2 -9682.489} C_VEL
LIN {X 0,Y 425.311,Z 59.503,A -85,B 0,C 180,E1 -9685.818,E2 -9685.818} C_VEL
LIN {X 0,Y 425.294,Z 59.508,A -85,B 0,C 180,E1 -9689.239,E2 -9689.239} C_VEL
LIN {X 0,Y 425.353,Z 59.5,A -85,B 0,C 180,E1 -9692.443,E2 -9692.443} C_VEL
LIN {X 0,Y 425.355,Z 59.497,A -85,B 0,C 180,E1 -9695.602,E2 -9695.602} C_VEL
LIN {X 0,Y 425.298,Z 59.511,A -85,B 0,C 180,E1 -9698.682,E2 -9698.682} C_VEL
LIN {X 0,Y 425.333,Z 59.5,A -85,B 0,C 180,E1 -9701.703,E2 -9701.703} C_VEL
LIN {X 0,Y 425.353,Z 59.501,A -85,B 0,C 180,E1 -9704.671,E2 -9704.671} C_VEL
LIN {X 0,Y 425.417,Z 59.49,A -85,B 0,C 180,E1 -9707.598,E2 -9707.598} C_VEL
LIN {X 0,Y 425.44,Z 59.487,A -85,B 0,C 180,E1 -9711.45,E2 -9711.45} C_VEL
LIN {X 0,Y 425.554,Z 59.476,A -85,B 0,C 180,E1 -9714.313,E2 -9714.313} C_VEL
LIN {X 0,Y 425.576,Z 59.474,A -85,B 0,C 180,E1 -9718.107,E2 -9718.107} C_VEL
LIN {X 0,Y 425.707,Z 59.459,A -85,B 0,C 180,E1 -9720,E2 -9720} C_VEL
LIN {X 0,Y 425.549,Z 59.473,A -85,B 0,C 180,E1 -9722.84,E2 -9722.84} C_VEL
LIN {X 0,Y 425.538,Z 59.481,A -85,B 0,C 180,E1 -9725.687,E2 -9725.687} C_VEL
LIN {X 0,Y 425.413,Z 59.49,A -85,B 0,C 180,E1 -9728.551,E2 -9728.551} C_VEL
LIN {X 0,Y 425.417,Z 59.489,A -85,B 0,C 180,E1 -9732.402,E2 -9732.402} C_VEL
LIN {X 0,Y 425.393,Z 59.492,A -85,B 0,C 180,E1 -9736.312,E2 -9736.312} C_VEL
LIN {X 0,Y 425.333,Z 59.502,A -85,B 0,C 180,E1 -9739.635,E2 -9739.635} C_VEL
LIN {X 0,Y 425.292,Z 59.505,A -85,B 0,C 180,E1 -9742.339,E2 -9742.339} C_VEL
LIN {X 0,Y 425.325,Z 59.504,A -85,B 0,C 180,E1 -9744.657,E2 -9744.657} C_VEL
LIN {X 0,Y 425.304,Z 59.504,A -85,B 0,C 180,E1 -9747.561,E2 -9747.561} C_VEL
LIN {X 0,Y 425.292,Z 59.511,A -85,B 0,C 180,E1 -9750.816,E2 -9750.816} C_VEL
LIN {X 0,Y 425.313,Z 59.506,A -85,B 0,C 180,E1 -9754.287,E2 -9754.287} C_VEL
LIN {X 0,Y 425.282,Z 59.506,A -85,B 0,C 180,E1 -9757.694,E2 -9757.694} C_VEL
LIN {X 0,Y 425.284,Z 59.512,A -85,B 0,C 180,E1 -9760.52,E2 -9760.52} C_VEL
LIN {X 0,Y 425.26,Z 59.509,A -85,B 0,C 180,E1 -9763.351,E2 -9763.351} C_VEL
LIN {X 0,Y 425.259,Z 59.511,A -85,B 0,C 180,E1 -9766.649,E2 -9766.649} C_VEL
LIN {X 0,Y 425.27,Z 59.513,A -85,B 0,C 180,E1 -9769.87,E2 -9769.87} C_VEL
LIN {X 0,Y 425.278,Z 59.508,A -85,B 0,C 180,E1 -9772.489,E2 -9772.489} C_VEL
LIN {X 0,Y 425.308,Z 59.51,A -85,B 0,C 180,E1 -9775.817,E2 -9775.817} C_VEL
LIN {X 0,Y 425.294,Z 59.507,A -85,B 0,C 180,E1 -9779.239,E2 -9779.239} C_VEL
LIN {X 0,Y 425.413,Z 59.557,A -85,B 0,C 180,E1 -9782.213,E2 -9782.213} C_VEL
LIN {X 0,Y 427.913,Z 72.358,A -85,B 0,C 180,E1 -9784.721,E2 -9784.721} C_VEL
LIN {X 0,Y 427.852,Z 77.992,A -85,B 0,C 180,E1 -9785.754,E2 -9785.754} C_VEL
LIN {X 0,Y 426.747,Z 97.54,A -85,B 0,C 180,E1 -9789.263,E2 -9789.263} C_VEL
LIN {X 0,Y 426.116,Z 110.556,A -85,B 0,C 180,E1 -9791.582,E2 -9791.582} C_VEL
LIN {X 0,Y 429.685,Z 137.971,A -85,B 0,C 180,E1 -9792.202,E2 -9792.202} C_VEL
LIN {X 0,Y 428.927,Z 219.494,A -85,B 0,C 180,E1 -9793.582,E2 -9793.582} C_VEL
LIN {X 0,Y 428.397,Z 232.822,A -85,B 0,C 180,E1 -9793.989,E2 -9793.989} C_VEL
LIN {X 0,Y 427.865,Z 245.632,A -85,B 0,C 180,E1 -9794.58,E2 -9794.58} C_VEL
LIN {X 0,Y 427.164,Z 257.789,A -85,B 0,C 180,E1 -9795.347,E2 -9795.347} C_VEL
LIN {X 0,Y 426.521,Z 269.392,A -85,B 0,C 180,E1 -9796.299,E2 -9796.299} C_VEL
LIN {X 0,Y 425.909,Z 279.85,A -85,B 0,C 180,E1 -9797.372,E2 -9797.372} C_VEL
LIN {X 0,Y 425.36,Z 289.208,A -85,B 0,C 180,E1 -9798.564,E2 -9798.564} C_VEL
LIN {X 0,Y 424.788,Z 298.289,A -85,B 0,C 180,E1 -9799.996,E2 -9799.996} C_VEL
LIN {X 0,Y 424.501,Z 305.609,A -85,B 0,C 180,E1 -9801.431,E2 -9801.431} C_VEL
LIN {X 0,Y 424.313,Z 311.451,A -85,B 0,C 180,E1 -9802.864,E2 -9802.864} C_VEL
LIN {X 0,Y 424.157,Z 316.037,A -85,B 0,C 180,E1 -9804.294,E2 -9804.294} C_VEL
LIN {X 0,Y 424.206,Z 318.457,A -85,B 0,C 180,E1 -9805.248,E2 -9805.248} C_VEL
LIN {X 0,Y 424.171,Z 320.432,A -85,B 0,C 180,E1 -9806.2,E2 -9806.2} C_VEL
LIN {X 0,Y 424.26,Z 321.995,A -85,B 0,C 180,E1 -9807.151,E2 -9807.151} C_VEL
LIN {X 0,Y 424.213,Z 323.095,A -85,B 0,C 180,E1 -9808.101,E2 -9808.101} C_VEL
LIN {X 0,Y 424.202,Z 323.785,A -85,B 0,C 180,E1 -9809.051,E2 -9809.051} C_VEL
LIN {X 0,Y 424.208,Z 324.087,A -85,B 0,C 180,E1 -9810,E2 -9810} C_VEL
LIN {X 0,Y 424.174,Z 323.998,A -85,B 0,C 180,E1 -9810.949,E2 -9810.949} C_VEL
LIN {X 0,Y 424.193,Z 323.487,A -85,B 0,C 180,E1 -9811.899,E2 -9811.899} C_VEL
LIN {X 0,Y 424.234,Z 322.564,A -85,B 0,C 180,E1 -9812.849,E2 -9812.849} C_VEL
LIN {X 0,Y 424.196,Z 319.516,A -85,B 0,C 180,E1 -9814.752,E2 -9814.752} C_VEL
LIN {X 0,Y 424.152,Z 316.043,A -85,B 0,C 180,E1 -9816.186,E2 -9816.186} C_VEL
LIN {X 0,Y 424.362,Z 311.524,A -85,B 0,C 180,E1 -9817.614,E2 -9817.614} C_VEL
LIN {X 0,Y 424.684,Z 304.688,A -85,B 0,C 180,E1 -9819.285,E2 -9819.285} C_VEL
LIN {X 0,Y 425.16,Z 297.283,A -85,B 0,C 180,E1 -9820.717,E2 -9820.717} C_VEL
LIN {X 0,Y 425.91,Z 288.12,A -85,B 0,C 180,E1 -9822.145,E2 -9822.145} C_VEL
LIN {X 0,Y 426.61,Z 277.749,A -85,B 0,C 180,E1 -9823.433,E2 -9823.433} C_VEL
LIN {X 0,Y 427.48,Z 266.828,A -85,B 0,C 180,E1 -9824.52,E2 -9824.52} C_VEL
LIN {X 0,Y 428.243,Z 256.458,A -85,B 0,C 180,E1 -9825.345,E2 -9825.345} C_VEL
LIN {X 0,Y 429.078,Z 244.038,A -85,B 0,C 180,E1 -9826.107,E2 -9826.107} C_VEL
LIN {X 0,Y 429.752,Z 232.496,A -85,B 0,C 180,E1 -9826.63,E2 -9826.63} C_VEL
LIN {X 0,Y 430.251,Z 219.36,A -85,B 0,C 180,E1 -9827.038,E2 -9827.038} C_VEL
LIN {X 0,Y 431.121,Z 137.523,A -85,B 0,C 180,E1 -9828.449,E2 -9828.449} C_VEL
LIN {X 0,Y 428.287,Z 118.79,A -85,B 0,C 180,E1 -9828.923,E2 -9828.923} C_VEL
LIN {X 0,Y 426.775,Z 110.187,A -85,B 0,C 180,E1 -9829.167,E2 -9829.167} C_VEL
LIN {X 0,Y 427.984,Z 90.952,A -85,B 0,C 180,E1 -9832.69,E2 -9832.69} C_VEL
LIN {X 0,Y 428.916,Z 77.381,A -85,B 0,C 180,E1 -9835.216,E2 -9835.216} C_VEL
LIN {X 0,Y 428.131,Z 71.953,A -85,B 0,C 180,E1 -9836.31,E2 -9836.31} C_VEL
LIN {X 0,Y 425.689,Z 61.122,A -85,B 0,C 180,E1 -9838.606,E2 -9838.606} C_VEL
LIN {X 0,Y 425.307,Z 59.505,A -85,B 0,C 180,E1 -9839.009,E2 -9839.009} C_VEL
LIN {X 0,Y 425.267,Z 59.513,A -85,B 0,C 180,E1 -9841.927,E2 -9841.927} C_VEL
LIN {X 0,Y 425.3,Z 59.507,A -85,B 0,C 180,E1 -9845.336,E2 -9845.336} C_VEL
LIN {X 0,Y 425.296,Z 59.501,A -85,B 0,C 180,E1 -9849.043,E2 -9849.043} C_VEL
LIN {X 0,Y 425.277,Z 59.506,A -85,B 0,C 180,E1 -9852.653,E2 -9852.653} C_VEL
LIN {X 0,Y 425.264,Z 59.509,A -85,B 0,C 180,E1 -9856.044,E2 -9856.044} C_VEL
LIN {X 0,Y 425.277,Z 59.505,A -85,B 0,C 180,E1 -9858.621,E2 -9858.621} C_VEL
LIN {X 0,Y 425.3,Z 59.503,A -85,B 0,C 180,E1 -9861.101,E2 -9861.101} C_VEL
LIN {X 0,Y 425.301,Z 59.504,A -85,B 0,C 180,E1 -9864.664,E2 -9864.664} C_VEL
LIN {X 0,Y 425.267,Z 59.509,A -85,B 0,C 180,E1 -9868.073,E2 -9868.073} C_VEL
LIN {X 0,Y 425.335,Z 59.504,A -85,B 0,C 180,E1 -9871.368,E2 -9871.368} C_VEL
LIN {X 0,Y 425.296,Z 59.504,A -85,B 0,C 180,E1 -9874.555,E2 -9874.555} C_VEL
LIN {X 0,Y 425.291,Z 59.503,A -85,B 0,C 180,E1 -9877.661,E2 -9877.661} C_VEL
LIN {X 0,Y 425.366,Z 59.502,A -85,B 0,C 180,E1 -9880.704,E2 -9880.704} C_VEL
LIN {X 0,Y 425.392,Z 59.489,A -85,B 0,C 180,E1 -9883.688,E2 -9883.688} C_VEL
LIN {X 0,Y 425.416,Z 59.486,A -85,B 0,C 180,E1 -9887.598,E2 -9887.598} C_VEL
LIN {X 0,Y 425.446,Z 59.487,A -85,B 0,C 180,E1 -9891.45,E2 -9891.45} C_VEL
LIN {X 0,Y 425.555,Z 59.476,A -85,B 0,C 180,E1 -9894.313,E2 -9894.313} C_VEL
LIN {X 0,Y 425.575,Z 59.468,A -85,B 0,C 180,E1 -9898.107,E2 -9898.107} C_VEL
LIN {X 0,Y 425.706,Z 59.459,A -85,B 0,C 180,E1 -9900,E2 -9900} C_VEL
LIN {X 0,Y 425.548,Z 59.471,A -85,B 0,C 180,E1 -9902.84,E2 -9902.84} C_VEL
LIN {X 0,Y 425.51,Z 59.479,A -85,B 0,C 180,E1 -9906.617,E2 -9906.617} C_VEL
LIN {X 0,Y 425.402,Z 59.491,A -85,B 0,C 180,E1 -9909.509,E2 -9909.509} C_VEL
LIN {X 0,Y 425.397,Z 59.495,A -85,B 0,C 180,E1 -9912.904,E2 -9912.904} C_VEL
LIN {X 0,Y 425.364,Z 59.499,A -85,B 0,C 180,E1 -9916.604,E2 -9916.604} C_VEL
LIN {X 0,Y 425.331,Z 59.501,A -85,B 0,C 180,E1 -9919.635,E2 -9919.635} C_VEL
LIN {X 0,Y 425.309,Z 59.504,A -85,B 0,C 180,E1 -9923.365,E2 -9923.365} C_VEL
LIN {X 0,Y 425.305,Z 59.507,A -85,B 0,C 180,E1 -9926.498,E2 -9926.498} C_VEL
LIN {X 0,Y 425.288,Z 59.506,A -85,B 0,C 180,E1 -9929.72,E2 -9929.72} C_VEL
LIN {X 0,Y 425.284,Z 59.507,A -85,B 0,C 180,E1 -9933.048,E2 -9933.048} C_VEL
LIN {X 0,Y 425.282,Z 59.51,A -85,B 0,C 180,E1 -9935.928,E2 -9935.928} C_VEL
LIN {X 0,Y 425.264,Z 59.51,A -85,B 0,C 180,E1 -9939.037,E2 -9939.037} C_VEL
LIN {X 0,Y 425.284,Z 59.504,A -85,B 0,C 180,E1 -9941.957,E2 -9941.957} C_VEL
LIN {X 0,Y 425.286,Z 59.509,A -85,B 0,C 180,E1 -9945.283,E2 -9945.283} C_VEL
LIN {X 0,Y 425.266,Z 59.511,A -85,B 0,C 180,E1 -9948.62,E2 -9948.62} C_VEL
LIN {X 0,Y 425.281,Z 59.509,A -85,B 0,C 180,E1 -9951.099,E2 -9951.099} C_VEL
LIN {X 0,Y 425.298,Z 59.509,A -85,B 0,C 180,E1 -9954.664,E2 -9954.664} C_VEL
LIN {X 0,Y 425.295,Z 59.515,A -85,B 0,C 180,E1 -9958.354,E2 -9958.354} C_VEL
LIN {X 0,Y 425.34,Z 59.605,A -85,B 0,C 180,E1 -9958.636,E2 -9958.636} C_VEL
LIN {X 0,Y 427.088,Z 68.392,A -85,B 0,C 180,E1 -9960.9,E2 -9960.9} C_VEL
LIN {X 0,Y 430.024,Z 78.095,A -85,B 0,C 180,E1 -9961.241,E2 -9961.241} C_VEL
LIN {X 0,Y 431.822,Z 85.566,A -85,B 0,C 180,E1 -9961.468,E2 -9961.468} C_VEL
LIN {X 0,Y 430.595,Z 175.228,A -85,B 0,C 180,E1 -9963.003,E2 -9963.003} C_VEL
LIN {X 0,Y 430.304,Z 188.816,A -85,B 0,C 180,E1 -9963.442,E2 -9963.442} C_VEL
LIN {X 0,Y 429.898,Z 201.388,A -85,B 0,C 180,E1 -9964.046,E2 -9964.046} C_VEL
LIN {X 0,Y 429.198,Z 213.097,A -85,B 0,C 180,E1 -9964.802,E2 -9964.802} C_VEL
LIN {X 0,Y 428.401,Z 224.857,A -85,B 0,C 180,E1 -9965.787,E2 -9965.787} C_VEL
LIN {X 0,Y 427.719,Z 234.288,A -85,B 0,C 180,E1 -9966.774,E2 -9966.774} C_VEL
LIN {X 0,Y 426.996,Z 243.873,A -85,B 0,C 180,E1 -9968.01,E2 -9968.01} C_VEL
LIN {X 0,Y 426.229,Z 253.047,A -85,B 0,C 180,E1 -9969.489,E2 -9969.489} C_VEL
LIN {X 0,Y 425.601,Z 260.372,A -85,B 0,C 180,E1 -9970.966,E2 -9970.966} C_VEL
LIN {X 0,Y 425.204,Z 265.268,A -85,B 0,C 180,E1 -9972.195,E2 -9972.195} C_VEL
LIN {X 0,Y 424.858,Z 269.979,A -85,B 0,C 180,E1 -9973.667,E2 -9973.667} C_VEL
LIN {X 0,Y 424.572,Z 273.528,A -85,B 0,C 180,E1 -9975.133,E2 -9975.133} C_VEL
LIN {X 0,Y 424.355,Z 276.027,A -85,B 0,C 180,E1 -9976.593,E2 -9976.593} C_VEL
LIN {X 0,Y 424.261,Z 277.334,A -85,B 0,C 180,E1 -9977.782,E2 -9977.782} C_VEL
LIN {X 0,Y 424.216,Z 277.76,A -85,B 0,C 180,E1 -9978.403,E2 -9978.403} C_VEL
LIN {X 0,Y 423.531,Z 278.184,A -85,B 0,C 180,E1 -9979.194,E2 -9979.194} C_VEL
LIN {X 0,Y 420.656,Z 278.307,A -85,B 0,C 180,E1 -9980.482,E2 -9980.482} C_VEL
LIN {X 0,Y 418.253,Z 277.818,A -85,B 0,C 180,E1 -9981.519,E2 -9981.519} C_VEL
LIN {X 0,Y 417.249,Z 277.093,A -85,B 0,C 180,E1 -9982.316,E2 -9982.316} C_VEL
LIN {X 0,Y 417.182,Z 276.739,A -85,B 0,C 180,E1 -9982.584,E2 -9982.584} C_VEL
LIN {X 0,Y 417.367,Z 274.228,A -85,B 0,C 180,E1 -9984.201,E2 -9984.201} C_VEL
LIN {X 0,Y 417.488,Z 270.886,A -85,B 0,C 180,E1 -9985.656,E2 -9985.656} C_VEL
LIN {X 0,Y 417.712,Z 266.478,A -85,B 0,C 180,E1 -9987.107,E2 -9987.107} C_VEL
LIN {X 0,Y 417.962,Z 260.895,A -85,B 0,C 180,E1 -9988.555,E2 -9988.555} C_VEL
LIN {X 0,Y 418.513,Z 253.884,A -85,B 0,C 180,E1 -9990,E2 -9990} C_VEL
LIN {X 0,Y 419.007,Z 245.172,A -85,B 0,C 180,E1 -9991.442,E2 -9991.442} C_VEL
LIN {X 0,Y 419.606,Z 235.281,A -85,B 0,C 180,E1 -9992.76,E2 -9992.76} C_VEL
LIN {X 0,Y 420.357,Z 225.138,A -85,B 0,C 180,E1 -9993.835,E2 -9993.835} C_VEL
LIN {X 0,Y 421.073,Z 213.906,A -85,B 0,C 180,E1 -9994.787,E2 -9994.787} C_VEL
LIN {X 0,Y 421.554,Z 202.318,A -85,B 0,C 180,E1 -9995.561,E2 -9995.561} C_VEL
LIN {X 0,Y 421.966,Z 189.665,A -85,B 0,C 180,E1 -9996.185,E2 -9996.185} C_VEL
LIN {X 0,Y 422.257,Z 176.214,A -85,B 0,C 180,E1 -9996.631,E2 -9996.631} C_VEL
LIN {X 0,Y 422.787,Z 134.25,A -85,B 0,C 180,E1 -9997.372,E2 -9997.372} C_VEL
LIN {X 0,Y 423.156,Z 85.193,A -85,B 0,C 180,E1 -9998.209,E2 -9998.209} C_VEL
LIN {X 0,Y 419.969,Z 69.49,A -85,B 0,C 180,E1 -9998.607,E2 -9998.607} C_VEL
LIN {X 0,Y 419.683,Z 68.211,A -85,B 0,C 180,E1 -9998.668,E2 -9998.668} C_VEL
LIN {X 0,Y 418.33,Z 60.379,A -85,B 0,C 180,E1 -10000.619,E2 -10000.619} C_VEL
LIN {X 0,Y 418.316,Z 60.375,A -85,B 0,C 180,E1 -10003.604,E2 -10003.604} C_VEL
LIN {X 0,Y 418.315,Z 60.378,A -85,B 0,C 180,E1 -10006.736,E2 -10006.736} C_VEL
LIN {X 0,Y 418.272,Z 60.381,A -85,B 0,C 180,E1 -10009.791,E2 -10009.791} C_VEL
LIN {X 0,Y 418.233,Z 60.386,A -85,B 0,C 180,E1 -10012.737,E2 -10012.737} C_VEL
LIN {X 0,Y 418.27,Z 60.384,A -85,B 0,C 180,E1 -10015.904,E2 -10015.904} C_VEL
LIN {X 0,Y 418.267,Z 60.38,A -85,B 0,C 180,E1 -10019.162,E2 -10019.162} C_VEL
LIN {X 0,Y 418.259,Z 60.381,A -85,B 0,C 180,E1 -10022.844,E2 -10022.844} C_VEL
LIN {X 0,Y 418.251,Z 60.384,A -85,B 0,C 180,E1 -10026.239,E2 -10026.239} C_VEL
LIN {X 0,Y 418.258,Z 60.388,A -85,B 0,C 180,E1 -10029.682,E2 -10029.682} C_VEL
LIN {X 0,Y 418.232,Z 60.385,A -85,B 0,C 180,E1 -10032.321,E2 -10032.321} C_VEL
LIN {X 0,Y 418.238,Z 60.387,A -85,B 0,C 180,E1 -10035.109,E2 -10035.109} C_VEL
LIN {X 0,Y 418.242,Z 60.386,A -85,B 0,C 180,E1 -10037.767,E2 -10037.767} C_VEL
LIN {X 0,Y 418.252,Z 60.383,A -85,B 0,C 180,E1 -10040.62,E2 -10040.62} C_VEL
LIN {X 0,Y 418.246,Z 60.383,A -85,B 0,C 180,E1 -10043.976,E2 -10043.976} C_VEL
LIN {X 0,Y 418.261,Z 60.386,A -85,B 0,C 180,E1 -10047.156,E2 -10047.156} C_VEL
LIN {X 0,Y 418.272,Z 60.387,A -85,B 0,C 180,E1 -10050.896,E2 -10050.896} C_VEL
LIN {X 0,Y 418.275,Z 60.38,A -85,B 0,C 180,E1 -10054.096,E2 -10054.096} C_VEL
LIN {X 0,Y 418.242,Z 60.384,A -85,B 0,C 180,E1 -10057.264,E2 -10057.264} C_VEL
LIN {X 0,Y 418.287,Z 60.382,A -85,B 0,C 180,E1 -10060.364,E2 -10060.364} C_VEL
LIN {X 0,Y 418.321,Z 60.373,A -85,B 0,C 180,E1 -10063.405,E2 -10063.405} C_VEL
LIN {X 0,Y 418.351,Z 60.37,A -85,B 0,C 180,E1 -10066.999,E2 -10066.999} C_VEL
LIN {X 0,Y 418.344,Z 60.376,A -85,B 0,C 180,E1 -10070.329,E2 -10070.329} C_VEL
LIN {X 0,Y 418.483,Z 60.353,A -85,B 0,C 180,E1 -10073.249,E2 -10073.249} C_VEL
LIN {X 0,Y 418.341,Z 60.371,A -85,B 0,C 180,E1 -10075.182,E2 -10075.182} C_VEL
LIN {X 0,Y 418.546,Z 60.351,A -85,B 0,C 180,E1 -10078.076,E2 -10078.076} C_VEL
LIN {X 0,Y 418.676,Z 60.334,A -85,B 0,C 180,E1 -10080,E2 -10080} C_VEL
LIN {X 0,Y 418.504,Z 60.351,A -85,B 0,C 180,E1 -10082.888,E2 -10082.888} C_VEL
LIN {X 0,Y 418.495,Z 60.357,A -85,B 0,C 180,E1 -10085.783,E2 -10085.783} C_VEL
LIN {X 0,Y 418.382,Z 60.366,A -85,B 0,C 180,E1 -10088.696,E2 -10088.696} C_VEL
LIN {X 0,Y 418.32,Z 60.378,A -85,B 0,C 180,E1 -10091.631,E2 -10091.631} C_VEL
LIN {X 0,Y 418.308,Z 60.375,A -85,B 0,C 180,E1 -10094.597,E2 -10094.597} C_VEL
LIN {X 0,Y 418.284,Z 60.381,A -85,B 0,C 180,E1 -10097.604,E2 -10097.604} C_VEL
LIN {X 0,Y 418.255,Z 60.384,A -85,B 0,C 180,E1 -10100.663,E2 -10100.663} C_VEL
LIN {X 0,Y 418.279,Z 60.379,A -85,B 0,C 180,E1 -10103.782,E2 -10103.782} C_VEL
LIN {X 0,Y 418.27,Z 60.384,A -85,B 0,C 180,E1 -10107.058,E2 -10107.058} C_VEL
LIN {X 0,Y 418.247,Z 60.384,A -85,B 0,C 180,E1 -10110.272,E2 -10110.272} C_VEL
LIN {X 0,Y 418.251,Z 60.382,A -85,B 0,C 180,E1 -10113.677,E2 -10113.677} C_VEL
LIN {X 0,Y 418.243,Z 60.384,A -85,B 0,C 180,E1 -10117.224,E2 -10117.224} C_VEL
LIN {X 0,Y 418.248,Z 60.383,A -85,B 0,C 180,E1 -10119.683,E2 -10119.683} C_VEL
LIN {X 0,Y 418.233,Z 60.391,A -85,B 0,C 180,E1 -10122.321,E2 -10122.321} C_VEL
LIN {X 0,Y 418.239,Z 60.384,A -85,B 0,C 180,E1 -10125.109,E2 -10125.109} C_VEL
LIN {X 0,Y 418.237,Z 60.387,A -85,B 0,C 180,E1 -10127.766,E2 -10127.766} C_VEL
LIN {X 0,Y 418.245,Z 60.385,A -85,B 0,C 180,E1 -10131.557,E2 -10131.557} C_VEL
LIN {X 0,Y 418.261,Z 60.381,A -85,B 0,C 180,E1 -10135.159,E2 -10135.159} C_VEL
LIN {X 0,Y 418.248,Z 60.386,A -85,B 0,C 180,E1 -10137.472,E2 -10137.472} C_VEL
LIN {X 0,Y 418.272,Z 60.385,A -85,B 0,C 180,E1 -10140.895,E2 -10140.895} C_VEL
LIN {X 0,Y 418.371,Z 60.423,A -85,B 0,C 180,E1 -10142.002,E2 -10142.002} C_VEL
LIN {X 0,Y 420.875,Z 73.299,A -85,B 0,C 180,E1 -10144.57,E2 -10144.57} C_VEL
LIN {X 0,Y 420.98,Z 77.344,A -85,B 0,C 180,E1 -10145.332,E2 -10145.332} C_VEL
LIN {X 0,Y 419.841,Z 96.9,A -85,B 0,C 180,E1 -10148.905,E2 -10148.905} C_VEL
LIN {X 0,Y 419.153,Z 110.27,A -85,B 0,C 180,E1 -10151.328,E2 -10151.328} C_VEL
LIN {X 0,Y 422.821,Z 138.615,A -85,B 0,C 180,E1 -10151.966,E2 -10151.966} C_VEL
LIN {X 0,Y 422.014,Z 219.772,A -85,B 0,C 180,E1 -10153.367,E2 -10153.367} C_VEL
LIN {X 0,Y 421.435,Z 233.65,A -85,B 0,C 180,E1 -10153.811,E2 -10153.811} C_VEL
LIN {X 0,Y 420.863,Z 246.624,A -85,B 0,C 180,E1 -10154.441,E2 -10154.441} C_VEL
LIN {X 0,Y 420.148,Z 258.442,A -85,B 0,C 180,E1 -10155.221,E2 -10155.221} C_VEL
LIN {X 0,Y 419.494,Z 269.855,A -85,B 0,C 180,E1 -10156.188,E2 -10156.188} C_VEL
LIN {X 0,Y 418.935,Z 279.339,A -85,B 0,C 180,E1 -10157.186,E2 -10157.186} C_VEL
LIN {X 0,Y 418.365,Z 288.541,A -85,B 0,C 180,E1 -10158.37,E2 -10158.37} C_VEL
LIN {X 0,Y 417.731,Z 297.668,A -85,B 0,C 180,E1 -10159.825,E2 -10159.825} C_VEL
LIN {X 0,Y 417.426,Z 305.032,A -85,B 0,C 180,E1 -10161.284,E2 -10161.284} C_VEL
LIN {X 0,Y 417.242,Z 310.922,A -85,B 0,C 180,E1 -10162.742,E2 -10162.742} C_VEL
LIN {X 0,Y 417.069,Z 315.543,A -85,B 0,C 180,E1 -10164.197,E2 -10164.197} C_VEL
LIN {X 0,Y 417.134,Z 317.985,A -85,B 0,C 180,E1 -10165.167,E2 -10165.167} C_VEL
LIN {X 0,Y 417.171,Z 321.551,A -85,B 0,C 180,E1 -10167.103,E2 -10167.103} C_VEL
LIN {X 0,Y 417.137,Z 322.678,A -85,B 0,C 180,E1 -10168.069,E2 -10168.069} C_VEL
LIN {X 0,Y 417.121,Z 323.695,A -85,B 0,C 180,E1 -10170,E2 -10170} C_VEL
LIN {X 0,Y 417.092,Z 323.619,A -85,B 0,C 180,E1 -10170.965,E2 -10170.965} C_VEL
LIN {X 0,Y 417.119,Z 323.135,A -85,B 0,C 180,E1 -10171.931,E2 -10171.931} C_VEL
LIN {X 0,Y 417.13,Z 322.224,A -85,B 0,C 180,E1 -10172.897,E2 -10172.897} C_VEL
LIN {X 0,Y 417.099,Z 319.203,A -85,B 0,C 180,E1 -10174.833,E2 -10174.833} C_VEL
LIN {X 0,Y 417.05,Z 316.14,A -85,B 0,C 180,E1 -10176.145,E2 -10176.145} C_VEL
LIN {X 0,Y 417.308,Z 311.273,A -85,B 0,C 180,E1 -10177.743,E2 -10177.743} C_VEL
LIN {X 0,Y 417.654,Z 304.491,A -85,B 0,C 180,E1 -10179.443,E2 -10179.443} C_VEL
LIN {X 0,Y 418.158,Z 297.129,A -85,B 0,C 180,E1 -10180.899,E2 -10180.899} C_VEL
LIN {X 0,Y 418.945,Z 288.027,A -85,B 0,C 180,E1 -10182.35,E2 -10182.35} C_VEL
LIN {X 0,Y 419.623,Z 278.613,A -85,B 0,C 180,E1 -10183.561,E2 -10183.561} C_VEL
LIN {X 0,Y 420.475,Z 268.192,A -85,B 0,C 180,E1 -10184.644,E2 -10184.644} C_VEL
LIN {X 0,Y 421.412,Z 256.641,A -85,B 0,C 180,E1 -10185.6,E2 -10185.6} C_VEL
LIN {X 0,Y 422.276,Z 244.463,A -85,B 0,C 180,E1 -10186.373,E2 -10186.373} C_VEL
LIN {X 0,Y 422.932,Z 233.214,A -85,B 0,C 180,E1 -10186.906,E2 -10186.906} C_VEL
LIN {X 0,Y 423.554,Z 219.49,A -85,B 0,C 180,E1 -10187.347,E2 -10187.347} C_VEL
LIN {X 0,Y 424.517,Z 138.613,A -85,B 0,C 180,E1 -10188.767,E2 -10188.767} C_VEL
LIN {X 0,Y 421.594,Z 119.312,A -85,B 0,C 180,E1 -10189.267,E2 -10189.267} C_VEL
LIN {X 0,Y 419.917,Z 109.714,A -85,B 0,C 180,E1 -10189.556,E2 -10189.556} C_VEL
LIN {X 0,Y 421.295,Z 88.954,A -85,B 0,C 180,E1 -10193.436,E2 -10193.436} C_VEL
LIN {X 0,Y 422.03,Z 78.635,A -85,B 0,C 180,E1 -10195.392,E2 -10195.392} C_VEL
LIN {X 0,Y 420.879,Z 71.866,A -85,B 0,C 180,E1 -10196.799,E2 -10196.799} C_VEL
LIN {X 0,Y 418.252,Z 60.384,A -85,B 0,C 180,E1 -10199.301,E2 -10199.301} C_VEL
LIN {X 0,Y 418.26,Z 60.385,A -85,B 0,C 180,E1 -10202.844,E2 -10202.844} C_VEL
LIN {X 0,Y 418.247,Z 60.387,A -85,B 0,C 180,E1 -10206.238,E2 -10206.238} C_VEL
LIN {X 0,Y 418.251,Z 60.378,A -85,B 0,C 180,E1 -10209.682,E2 -10209.682} C_VEL
LIN {X 0,Y 418.233,Z 60.384,A -85,B 0,C 180,E1 -10212.321,E2 -10212.321} C_VEL
LIN {X 0,Y 418.238,Z 60.382,A -85,B 0,C 180,E1 -10215.109,E2 -10215.109} C_VEL
LIN {X 0,Y 418.243,Z 60.384,A -85,B 0,C 180,E1 -10217.767,E2 -10217.767} C_VEL
LIN {X 0,Y 418.248,Z 60.378,A -85,B 0,C 180,E1 -10220.621,E2 -10220.621} C_VEL
LIN {X 0,Y 418.246,Z 60.383,A -85,B 0,C 180,E1 -10223.976,E2 -10223.976} C_VEL
LIN {X 0,Y 418.26,Z 60.383,A -85,B 0,C 180,E1 -10227.156,E2 -10227.156} C_VEL
LIN {X 0,Y 418.272,Z 60.381,A -85,B 0,C 180,E1 -10230.895,E2 -10230.895} C_VEL
LIN {X 0,Y 418.273,Z 60.376,A -85,B 0,C 180,E1 -10234.096,E2 -10234.096} C_VEL
LIN {X 0,Y 418.242,Z 60.383,A -85,B 0,C 180,E1 -10237.264,E2 -10237.264} C_VEL
LIN {X 0,Y 418.287,Z 60.381,A -85,B 0,C 180,E1 -10240.364,E2 -10240.364} C_VEL
